C05361=1026.292,340.312,-136.892,171.555,47.662,159.342
C05362=1026.299,340.560,-136.929,171.561,47.662,159.342
C05363=1026.307,340.806,-136.966,171.568,47.662,159.343
C05364=1026.314,341.053,-137.002,171.574,47.662,159.344
C05365=1026.322,341.300,-137.038,171.581,47.662,159.345
C05366=1026.329,341.548,-137.075,171.586,47.662,159.346
C05367=1026.336,341.795,-137.111,171.593,47.661,159.347
C05368=1026.344,342.042,-137.148,171.599,47.662,159.347
C05369=1026.351,342.290,-137.185,171.606,47.661,159.348
C05370=1026.359,342.537,-137.222,171.612,47.662,159.349
C05371=1026.366,342.784,-137.259,171.618,47.661,159.350
C05372=1026.374,343.031,-137.296,171.624,47.662,159.351
C05373=1026.382,343.279,-137.332,171.631,47.662,159.352
C05374=1026.388,343.525,-137.369,171.637,47.662,159.352
C05375=1026.396,343.772,-137.405,171.644,47.662,159.353
C05376=1026.404,344.019,-137.442,171.650,47.661,159.354
C05377=1026.411,344.266,-137.480,171.657,47.662,159.355
C05378=1026.419,344.514,-137.516,171.663,47.662,159.356
C05379=1026.426,344.761,-137.554,171.669,47.661,159.357
C05380=1026.434,345.008,-137.591,171.675,47.662,159.358
C05381=1026.441,345.256,-137.627,171.682,47.662,159.359
C05382=1026.450,345.503,-137.665,171.688,47.662,159.360
C05383=1026.458,345.750,-137.702,171.695,47.662,159.360
C05384=1026.465,345.997,-137.739,171.702,47.662,159.361
C05385=1026.473,346.244,-137.776,171.708,47.662,159.362
C05386=1026.480,346.492,-137.813,171.715,47.662,159.363
C05387=1026.488,346.739,-137.850,171.721,47.663,159.364
C05388=1026.495,346.986,-137.887,171.728,47.662,159.365
C05389=1026.503,347.232,-137.924,171.735,47.662,159.366
C05390=1026.510,347.480,-137.962,171.741,47.663,159.367
C05391=1026.519,347.727,-137.999,171.748,47.663,159.368
C05392=1026.527,347.974,-138.036,171.754,47.663,159.369
C05393=1026.534,348.221,-138.074,171.761,47.663,159.370
C05394=1026.541,348.468,-138.111,171.768,47.664,159.371
C05395=1026.549,348.715,-138.148,171.774,47.664,159.371
C05396=1026.557,348.962,-138.186,171.781,47.664,159.372
C05397=1026.564,349.210,-138.223,171.787,47.664,159.373
C05398=1026.573,349.456,-138.261,171.794,47.665,159.374
C05399=1026.580,349.703,-138.299,171.801,47.665,159.375
C05400=1026.587,349.950,-138.336,171.807,47.665,159.376
C05401=1026.595,350.197,-138.373,171.814,47.666,159.377
C05402=1026.602,350.418,-138.407,171.820,47.666,159.378
C05403=1026.609,350.638,-138.441,171.826,47.666,159.379
C05404=1026.616,350.859,-138.475,171.832,47.666,159.380
C05405=1026.622,351.080,-138.508,171.838,47.667,159.381
C05406=1026.630,351.301,-138.542,171.844,47.667,159.382
C05407=1026.636,351.521,-138.576,171.850,47.667,159.383
C05408=1026.644,351.742,-138.609,171.856,47.668,159.383
C05409=1026.650,351.962,-138.643,171.863,47.668,159.384
C05410=1026.658,352.210,-138.681,171.869,47.668,159.385
C05411=1026.667,352.456,-138.719,171.876,47.668,159.386
C05412=1026.674,352.704,-138.757,171.883,47.669,159.387
C05413=1026.682,352.950,-138.795,171.889,47.669,159.388
C05414=1026.690,353.197,-138.832,171.896,47.670,159.389
C05415=1026.698,353.444,-138.870,171.903,47.670,159.390
C05416=1026.705,353.691,-138.908,171.910,47.670,159.391
C05417=1026.714,353.938,-138.946,171.916,47.671,159.392
C05418=1026.722,354.185,-138.984,171.924,47.671,159.393
C05419=1026.730,354.433,-139.022,171.931,47.672,159.394
C05420=1026.737,354.679,-139.060,171.938,47.672,159.396
C05421=1026.746,354.926,-139.098,171.944,47.673,159.396
C05422=1026.753,355.173,-139.136,171.951,47.673,159.398
C05423=1026.761,355.420,-139.175,171.959,47.674,159.399
C05424=1026.769,355.667,-139.213,171.966,47.674,159.400
C05425=1026.777,355.914,-139.251,171.972,47.675,159.401
C05426=1026.785,356.161,-139.290,171.979,47.675,159.402
C05427=1026.793,356.408,-139.328,171.986,47.676,159.403
C05428=1026.800,356.654,-139.366,171.994,47.677,159.404
C05429=1026.809,356.902,-139.405,172.001,47.677,159.405
C05430=1026.816,357.149,-139.443,172.008,47.677,159.406
C05431=1026.824,357.396,-139.481,172.014,47.678,159.407
C05432=1026.833,357.643,-139.519,172.022,47.679,159.409
C05433=1026.841,357.889,-139.558,172.029,47.680,159.410
C05434=1026.849,358.136,-139.597,172.036,47.680,159.411
C05435=1026.857,358.383,-139.635,172.043,47.680,159.412
C05436=1026.865,358.630,-139.674,172.051,47.681,159.413
C05437=1026.873,358.877,-139.712,172.057,47.682,159.414
C05438=1026.881,359.124,-139.751,172.064,47.683,159.415
C05439=1026.888,359.371,-139.789,172.072,47.684,159.416
C05440=1026.897,359.617,-139.828,172.079,47.684,159.418
C05441=1026.905,359.864,-139.867,172.086,47.685,159.419
C05442=1026.913,360.111,-139.905,172.094,47.686,159.420
C05443=1026.921,360.358,-139.944,172.101,47.686,159.421
C05444=1026.929,360.605,-139.983,172.108,47.687,159.422
C05445=1026.937,360.852,-140.022,172.116,47.688,159.423
C05446=1026.944,361.098,-140.061,172.123,47.688,159.424
C05447=1026.953,361.345,-140.100,172.129,47.689,159.426
C05448=1026.961,361.592,-140.139,172.137,47.690,159.427
C05449=1026.969,361.839,-140.178,172.144,47.691,159.428
C05450=1026.977,362.086,-140.218,172.152,47.692,159.429
C05451=1026.985,362.332,-140.257,172.159,47.693,159.430
C05452=1026.993,362.579,-140.295,172.166,47.693,159.432
C05453=1027.001,362.826,-140.335,172.174,47.695,159.433
C05454=1027.009,363.073,-140.374,172.181,47.695,159.434
C05455=1027.017,363.320,-140.413,172.189,47.696,159.435
C05456=1027.026,363.567,-140.453,172.196,47.697,159.437
C05457=1027.034,363.813,-140.492,172.203,47.698,159.438
C05458=1027.042,364.061,-140.531,172.211,47.699,159.439
C05459=1027.050,364.307,-140.570,172.218,47.700,159.440
C05460=1027.058,364.553,-140.609,172.226,47.700,159.441
C05461=1027.066,364.800,-140.649,172.233,47.702,159.443
C05462=1027.073,365.024,-140.685,172.241,47.702,159.444
C05463=1027.081,365.248,-140.720,172.247,47.703,159.445
C05464=1027.088,365.472,-140.756,172.254,47.704,159.446
C05465=1027.096,365.696,-140.792,172.261,47.705,159.447
C05466=1027.103,365.920,-140.828,172.268,47.706,159.448
C05467=1027.111,366.144,-140.863,172.274,47.707,159.449
C05468=1027.119,366.367,-140.899,172.282,47.708,159.451
C05469=1027.126,366.591,-140.935,172.288,47.709,159.452
C05470=1027.134,366.838,-140.974,172.296,47.710,159.453
C05471=1027.143,367.084,-141.014,172.303,47.711,159.454
C05472=1027.152,367.332,-141.055,172.311,47.712,159.456
C05473=1027.160,367.578,-141.094,172.319,47.712,159.457
C05474=1027.168,367.825,-141.133,172.327,47.714,159.458
C05475=1027.177,368.071,-141.173,172.335,47.715,159.460
C05476=1027.185,368.318,-141.213,172.342,47.716,159.461
C05477=1027.193,368.564,-141.253,172.350,47.717,159.462
C05478=1027.202,368.812,-141.292,172.357,47.718,159.464
C05479=1027.210,369.058,-141.332,172.366,47.719,159.465
C05480=1027.219,369.304,-141.372,172.374,47.720,159.466
C05481=1027.227,369.551,-141.412,172.381,47.722,159.468
C05482=1027.235,369.798,-141.453,172.389,47.723,159.469
C05483=1027.244,370.045,-141.493,172.397,47.724,159.470
C05484=1027.252,370.291,-141.533,172.404,47.725,159.472
C05485=1027.260,370.538,-141.573,172.413,47.726,159.473
C05486=1027.268,370.784,-141.613,172.421,47.728,159.475
C05487=1027.277,371.032,-141.653,172.428,47.729,159.476
C05488=1027.285,371.278,-141.694,172.436,47.731,159.477
C05489=1027.293,371.524,-141.734,172.444,47.732,159.479
C05490=1027.303,371.771,-141.775,172.452,47.733,159.480
C05491=1027.310,372.018,-141.814,172.460,47.734,159.482
C05492=1027.319,372.264,-141.855,172.468,47.735,159.483
C05493=1027.328,372.511,-141.896,172.476,47.737,159.484
C05494=1027.336,372.757,-141.936,172.484,47.738,159.486
C05495=1027.344,373.003,-141.975,172.492,47.739,159.487
C05496=1027.353,373.250,-142.016,172.500,47.741,159.489
C05497=1027.361,373.497,-142.057,172.509,47.742,159.490
C05498=1027.370,373.743,-142.098,172.516,47.743,159.492
C05499=1027.378,373.990,-142.138,172.524,47.745,159.493
C05500=1027.388,374.236,-142.179,172.533,47.746,159.495
C05501=1027.396,374.483,-142.219,172.541,47.747,159.496
C05502=1027.404,374.730,-142.260,172.549,47.749,159.497
C05503=1027.413,374.976,-142.300,172.557,47.750,159.499
C05504=1027.422,375.223,-142.341,172.565,47.752,159.500
C05505=1027.431,375.468,-142.381,172.573,47.753,159.502
C05506=1027.439,375.715,-142.423,172.582,47.755,159.503
C05507=1027.448,375.962,-142.464,172.590,47.757,159.505
C05508=1027.457,376.208,-142.504,172.599,47.758,159.506
C05509=1027.465,376.455,-142.545,172.607,47.759,159.508
C05510=1027.475,376.701,-142.585,172.616,47.761,159.510
C05511=1027.483,376.947,-142.627,172.623,47.762,159.511
C05512=1027.492,377.194,-142.668,172.631,47.764,159.512
C05513=1027.500,377.441,-142.709,172.640,47.766,159.514
C05514=1027.509,377.687,-142.750,172.648,47.767,159.516
C05515=1027.518,377.933,-142.792,172.657,47.769,159.517
C05516=1027.526,378.180,-142.833,172.665,47.771,159.519
C05517=1027.535,378.426,-142.874,172.674,47.772,159.520
C05518=1027.544,378.672,-142.915,172.682,47.773,159.522
C05519=1027.553,378.919,-142.956,172.691,47.775,159.523
C05520=1027.561,379.164,-142.998,172.699,47.777,159.525
C05521=1027.570,379.411,-143.039,172.708,47.778,159.527
C05522=1027.578,379.636,-143.077,172.716,47.780,159.528
C05523=1027.586,379.862,-143.115,172.724,47.782,159.530
C05524=1027.594,380.087,-143.152,172.731,47.783,159.531
C05525=1027.602,380.312,-143.191,172.739,47.785,159.533
C05526=1027.610,380.537,-143.229,172.747,47.786,159.534
C05527=1027.618,380.762,-143.266,172.755,47.788,159.535
C05528=1027.626,380.987,-143.305,172.763,47.790,159.537
C05529=1027.634,381.213,-143.343,172.771,47.791,159.538
C05530=1027.643,381.458,-143.384,172.779,47.793,159.540
C05531=1027.651,381.705,-143.426,172.788,47.795,159.542
C05532=1027.660,381.951,-143.467,172.796,47.797,159.543
C05533=1027.669,382.197,-143.509,172.805,47.799,159.545
C05534=1027.679,382.443,-143.550,172.814,47.800,159.547
C05535=1027.688,382.690,-143.592,172.822,47.802,159.548
C05536=1027.697,382.936,-143.634,172.832,47.804,159.550
C05537=1027.706,383.182,-143.676,172.841,47.806,159.552
C05538=1027.715,383.428,-143.718,172.849,47.808,159.553
C05539=1027.724,383.675,-143.760,172.858,47.810,159.555
C05540=1027.733,383.921,-143.801,172.867,47.812,159.557
C05541=1027.743,384.168,-143.844,172.876,47.813,159.559
C05542=1027.752,384.414,-143.886,172.885,47.816,159.560
C05543=1027.761,384.660,-143.928,172.894,47.817,159.562
C05544=1027.770,384.906,-143.970,172.903,47.819,159.564
C05545=1027.779,385.152,-144.012,172.912,47.821,159.566
C05546=1027.788,385.399,-144.053,172.920,47.823,159.567
C05547=1027.797,385.644,-144.096,172.930,47.825,159.569
C05548=1027.807,385.892,-144.138,172.939,47.827,159.571
C05549=1027.816,386.137,-144.180,172.948,47.829,159.573
C05550=1027.825,386.384,-144.222,172.957,47.831,159.574
C05551=1027.834,386.629,-144.264,172.967,47.833,159.576
C05552=1027.844,386.876,-144.307,172.975,47.835,159.578
C05553=1027.852,387.122,-144.350,172.984,47.837,159.580
C05554=1027.862,387.387,-144.395,172.995,47.840,159.582
C05555=1027.872,387.652,-144.442,173.004,47.842,159.583
C05556=1027.882,387.917,-144.487,173.014,47.844,159.585
C05557=1027.892,388.182,-144.533,173.025,47.847,159.588
C05558=1027.902,388.428,-144.576,173.034,47.849,159.589
C05559=1027.911,388.674,-144.618,173.043,47.851,159.591
C05560=1027.919,388.920,-144.661,173.053,47.853,159.593
C05561=1027.929,389.166,-144.704,173.061,47.855,159.595
C05562=1027.939,389.412,-144.747,173.070,47.857,159.597
C05563=1027.948,389.658,-144.789,173.080,47.860,159.599
C05564=1027.957,389.904,-144.832,173.089,47.862,159.600
C05565=1027.967,390.151,-144.875,173.099,47.864,159.602
C05566=1027.975,390.397,-144.918,173.108,47.867,159.604
C05567=1027.985,390.642,-144.961,173.118,47.869,159.606
C05568=1027.995,390.889,-145.004,173.127,47.871,159.608
C05569=1028.004,391.135,-145.048,173.137,47.873,159.610
C05570=1028.013,391.381,-145.090,173.146,47.876,159.612
C05571=1028.022,391.627,-145.134,173.156,47.878,159.614
C05572=1028.032,391.873,-145.177,173.165,47.881,159.616
C05573=1028.042,392.119,-145.220,173.176,47.882,159.618
C05574=1028.050,392.365,-145.263,173.185,47.885,159.620
C05575=1028.060,392.611,-145.307,173.195,47.888,159.622
C05576=1028.070,392.857,-145.350,173.205,47.890,159.624
C05577=1028.079,393.103,-145.393,173.214,47.892,159.626
C05578=1028.089,393.349,-145.436,173.224,47.895,159.628
C05579=1028.098,393.595,-145.480,173.233,47.897,159.630
C05580=1028.108,393.841,-145.524,173.243,47.900,159.632
C05581=1028.117,394.086,-145.567,173.254,47.902,159.634
C05582=1028.127,394.346,-145.613,173.263,47.905,159.636
C05583=1028.137,394.604,-145.659,173.274,47.907,159.638
C05584=1028.148,394.864,-145.705,173.284,47.910,159.640
C05585=1028.157,395.122,-145.751,173.295,47.913,159.642
C05586=1028.168,395.368,-145.795,173.304,47.915,159.644
C05587=1028.176,395.614,-145.839,173.314,47.918,159.646
C05588=1028.187,395.859,-145.882,173.325,47.921,159.648
C05589=1028.196,396.106,-145.926,173.335,47.923,159.650
C05590=1028.205,396.352,-145.970,173.345,47.926,159.653
C05591=1028.216,396.598,-146.014,173.355,47.928,159.655
C05592=1028.225,396.844,-146.058,173.365,47.931,159.657
C05593=1028.235,397.090,-146.102,173.375,47.934,159.659
C05594=1028.245,397.335,-146.146,173.386,47.936,159.661
C05595=1028.255,397.581,-146.190,173.395,47.939,159.663
C05596=1028.264,397.827,-146.234,173.405,47.942,159.665
C05597=1028.274,398.073,-146.278,173.416,47.944,159.667
C05598=1028.284,398.318,-146.322,173.426,47.947,159.670
C05599=1028.294,398.564,-146.366,173.437,47.950,159.672
C05600=1028.303,398.810,-146.411,173.447,47.953,159.674
C05601=1028.313,399.056,-146.455,173.456,47.955,159.676
C05602=1028.323,399.301,-146.500,173.467,47.958,159.678
C05603=1028.333,399.547,-146.544,173.477,47.961,159.680
C05604=1028.343,399.794,-146.589,173.488,47.964,159.683
C05605=1028.353,400.039,-146.633,173.498,47.967,159.685
C05606=1028.363,400.284,-146.678,173.509,47.970,159.687
C05607=1028.372,400.531,-146.722,173.519,47.973,159.689
C05608=1028.382,400.776,-146.767,173.530,47.976,159.692
C05609=1028.393,401.022,-146.812,173.540,47.979,159.694
C05610=1028.403,401.267,-146.856,173.551,47.982,159.696
C05611=1028.413,401.513,-146.901,173.561,47.985,159.698
C05612=1028.422,401.758,-146.946,173.572,47.988,159.701
C05613=1028.433,402.005,-146.991,173.583,47.990,159.703
C05614=1028.442,402.250,-147.036,173.593,47.994,159.705
C05615=1028.452,402.496,-147.081,173.604,47.996,159.707
C05616=1028.462,402.742,-147.126,173.614,47.999,159.710
C05617=1028.472,402.987,-147.171,173.625,48.002,159.712
C05618=1028.483,403.233,-147.217,173.637,48.006,159.714
C05619=1028.493,403.479,-147.262,173.647,48.009,159.717
C05620=1028.502,403.724,-147.306,173.658,48.012,159.719
C05621=1028.513,403.970,-147.352,173.669,48.015,159.721
C05622=1028.523,404.215,-147.397,173.680,48.018,159.724
C05623=1028.533,404.461,-147.442,173.691,48.021,159.726
C05624=1028.543,404.706,-147.488,173.702,48.024,159.729
C05625=1028.553,404.952,-147.533,173.713,48.028,159.731
C05626=1028.564,405.198,-147.579,173.724,48.030,159.733
C05627=1028.574,405.444,-147.624,173.734,48.034,159.736
C05628=1028.584,405.689,-147.670,173.746,48.037,159.738
C05629=1028.594,405.934,-147.715,173.757,48.040,159.741
C05630=1028.605,406.180,-147.760,173.768,48.044,159.743
C05631=1028.615,406.426,-147.806,173.780,48.047,159.746
C05632=1028.626,406.671,-147.852,173.791,48.050,159.748
C05633=1028.636,406.917,-147.897,173.802,48.053,159.750
C05634=1028.646,407.163,-147.943,173.813,48.056,159.753
C05635=1028.657,407.408,-147.989,173.825,48.060,159.755
C05636=1028.667,407.654,-148.035,173.836,48.063,159.758
C05637=1028.678,407.899,-148.081,173.848,48.066,159.760
C05638=1028.687,408.145,-148.127,173.859,48.070,159.763
C05639=1028.698,408.390,-148.173,173.870,48.073,159.765
C05640=1028.709,408.636,-148.219,173.882,48.076,159.768
C05641=1028.719,408.881,-148.265,173.893,48.080,159.770
C05642=1028.732,409.163,-148.317,173.906,48.084,159.773
C05643=1028.744,409.442,-148.370,173.919,48.088,159.776
C05644=1028.756,409.723,-148.422,173.932,48.092,159.779
C05645=1028.769,410.004,-148.475,173.946,48.095,159.782
C05646=1028.780,410.249,-148.521,173.958,48.099,159.785
C05647=1028.789,410.495,-148.568,173.969,48.103,159.787
C05648=1028.800,410.740,-148.614,173.981,48.107,159.790
C05649=1028.810,410.986,-148.661,173.992,48.110,159.793
C05650=1028.821,411.231,-148.708,174.005,48.113,159.795
C05651=1028.832,411.477,-148.754,174.017,48.117,159.798
C05652=1028.842,411.722,-148.801,174.028,48.121,159.801
C05653=1028.853,411.967,-148.847,174.040,48.124,159.803
C05654=1028.865,412.213,-148.894,174.052,48.128,159.806
C05655=1028.874,412.458,-148.941,174.064,48.132,159.809
C05656=1028.885,412.703,-148.987,174.076,48.136,159.812
C05657=1028.896,412.948,-149.034,174.088,48.140,159.814
C05658=1028.907,413.194,-149.082,174.101,48.143,159.817
C05659=1028.918,413.439,-149.128,174.112,48.147,159.820
C05660=1028.928,413.685,-149.175,174.125,48.150,159.823
C05661=1028.940,413.930,-149.222,174.137,48.154,159.825
C05662=1028.951,414.175,-149.269,174.149,48.158,159.828
C05663=1028.961,414.421,-149.317,174.161,48.162,159.831
C05664=1028.972,414.666,-149.363,174.173,48.165,159.834
C05665=1028.984,414.912,-149.410,174.186,48.169,159.836
C05666=1028.994,415.157,-149.458,174.198,48.173,159.839
C05667=1029.006,415.402,-149.505,174.211,48.177,159.842
C05668=1029.017,415.647,-149.552,174.223,48.181,159.845
C05669=1029.028,415.893,-149.600,174.235,48.185,159.848
C05670=1029.039,416.138,-149.647,174.248,48.188,159.851
C05671=1029.050,416.384,-149.694,174.260,48.193,159.854
C05672=1029.061,416.629,-149.742,174.273,48.197,159.857
C05673=1029.072,416.873,-149.790,174.285,48.200,159.859
C05674=1029.083,417.119,-149.838,174.298,48.205,159.862
C05675=1029.095,417.364,-149.885,174.311,48.209,159.865
C05676=1029.105,417.609,-149.933,174.323,48.213,159.868
C05677=1029.117,417.854,-149.981,174.337,48.217,159.871
C05678=1029.128,418.099,-150.029,174.350,48.221,159.874
C05679=1029.139,418.345,-150.077,174.362,48.224,159.877
C05680=1029.150,418.590,-150.124,174.375,48.229,159.880
C05681=1029.161,418.835,-150.172,174.388,48.233,159.883
C05682=1029.172,419.080,-150.221,174.401,48.237,159.886
C05683=1029.184,419.325,-150.268,174.414,48.241,159.889
C05684=1029.196,419.570,-150.317,174.427,48.245,159.892
C05685=1029.207,419.816,-150.366,174.440,48.249,159.895
C05686=1029.218,420.061,-150.413,174.454,48.254,159.898
C05687=1029.230,420.306,-150.462,174.467,48.258,159.901
C05688=1029.242,420.550,-150.510,174.479,48.262,159.904
C05689=1029.253,420.796,-150.558,174.493,48.267,159.908
C05690=1029.264,421.041,-150.607,174.506,48.271,159.911
C05691=1029.276,421.286,-150.655,174.520,48.275,159.914
C05692=1029.287,421.531,-150.703,174.533,48.279,159.917
C05693=1029.299,421.776,-150.752,174.547,48.284,159.920
C05694=1029.310,422.021,-150.800,174.560,48.288,159.923
C05695=1029.322,422.266,-150.850,174.574,48.293,159.927
C05696=1029.333,422.512,-150.898,174.587,48.297,159.930
C05697=1029.345,422.756,-150.947,174.600,48.301,159.933
C05698=1029.357,423.001,-150.995,174.614,48.306,159.936
C05699=1029.369,423.246,-151.045,174.628,48.310,159.939
C05700=1029.380,423.491,-151.094,174.642,48.314,159.943
C05701=1029.392,423.736,-151.143,174.655,48.319,159.946
C05702=1029.406,424.027,-151.201,174.672,48.325,159.950
C05703=1029.420,424.318,-151.260,174.688,48.330,159.954
C05704=1029.434,424.609,-151.318,174.704,48.335,159.957
C05705=1029.448,424.900,-151.376,174.721,48.341,159.961
C05706=1029.460,425.145,-151.425,174.736,48.345,159.965
C05707=1029.472,425.390,-151.475,174.749,48.350,159.968
C05708=1029.483,425.634,-151.525,174.764,48.355,159.972
C05709=1029.495,425.880,-151.574,174.777,48.359,159.975
C05710=1029.508,426.123,-151.623,174.792,48.364,159.978
C05711=1029.520,426.369,-151.672,174.806,48.369,159.982
C05712=1029.532,426.614,-151.722,174.821,48.373,159.985
C05713=1029.543,426.858,-151.772,174.834,48.378,159.989
C05714=1029.556,427.103,-151.822,174.849,48.383,159.992
C05715=1029.567,427.348,-151.872,174.863,48.388,159.995
C05716=1029.579,427.592,-151.922,174.878,48.392,159.999
C05717=1029.591,427.838,-151.971,174.893,48.397,160.002
C05718=1029.603,428.083,-152.022,174.907,48.402,160.006
C05719=1029.616,428.328,-152.072,174.921,48.407,160.009
C05720=1029.627,428.572,-152.121,174.937,48.412,160.013
C05721=1029.640,428.816,-152.171,174.952,48.416,160.017
C05722=1029.652,429.061,-152.222,174.965,48.421,160.020
C05723=1029.665,429.306,-152.272,174.981,48.427,160.024
C05724=1029.676,429.551,-152.323,174.995,48.431,160.027
C05725=1029.688,429.795,-152.373,175.011,48.436,160.031
C05726=1029.701,430.040,-152.424,175.025,48.441,160.035
C05727=1029.713,430.284,-152.474,175.041,48.446,160.038
C05728=1029.726,430.529,-152.525,175.056,48.451,160.042
C05729=1029.738,430.774,-152.575,175.071,48.456,160.046
C05730=1029.751,431.018,-152.626,175.086,48.461,160.049
C05731=1029.763,431.263,-152.676,175.101,48.466,160.053
C05732=1029.776,431.507,-152.727,175.116,48.471,160.057
C05733=1029.789,431.751,-152.777,175.132,48.477,160.060
C05734=1029.801,431.996,-152.828,175.147,48.482,160.064
C05735=1029.813,432.241,-152.879,175.162,48.487,160.068
C05736=1029.826,432.485,-152.930,175.178,48.492,160.072
C05737=1029.839,432.729,-152.981,175.193,48.497,160.075
C05738=1029.852,432.974,-153.032,175.209,48.502,160.079
C05739=1029.864,433.218,-153.083,175.225,48.507,160.083
C05740=1029.878,433.463,-153.134,175.240,48.512,160.087
C05741=1029.890,433.708,-153.185,175.256,48.518,160.091
C05742=1029.902,433.952,-153.236,175.272,48.523,160.095
C05743=1029.915,434.197,-153.287,175.288,48.528,160.099
C05744=1029.928,434.441,-153.339,175.304,48.534,160.103
C05745=1029.941,434.686,-153.391,175.320,48.539,160.106
C05746=1029.954,434.929,-153.442,175.335,48.544,160.110
C05747=1029.967,435.174,-153.493,175.352,48.550,160.114
C05748=1029.980,435.418,-153.545,175.367,48.555,160.118
C05749=1029.993,435.662,-153.598,175.384,48.561,160.122
C05750=1030.006,435.907,-153.649,175.401,48.566,160.126
C05751=1030.019,436.151,-153.700,175.416,48.571,160.130
C05752=1030.032,436.396,-153.753,175.433,48.577,160.134
C05753=1030.045,436.640,-153.805,175.450,48.582,160.138
C05754=1030.057,436.884,-153.857,175.465,48.588,160.142
C05755=1030.071,437.128,-153.909,175.482,48.594,160.147
C05756=1030.084,437.372,-153.961,175.499,48.599,160.151
C05757=1030.097,437.617,-154.013,175.516,48.605,160.155
C05758=1030.111,437.861,-154.065,175.533,48.611,160.159
C05759=1030.123,438.104,-154.118,175.550,48.616,160.163
C05760=1030.137,438.349,-154.170,175.566,48.622,160.167
C05761=1030.150,438.593,-154.222,175.582,48.628,160.172
C05762=1030.165,438.860,-154.279,175.602,48.633,160.176
C05763=1030.179,439.127,-154.337,175.620,48.640,160.181
C05764=1030.195,439.394,-154.395,175.639,48.646,160.186
C05765=1030.208,439.660,-154.452,175.657,48.652,160.190
C05766=1030.223,439.905,-154.505,175.675,48.658,160.195
C05767=1030.236,440.149,-154.557,175.692,48.664,160.199
C05768=1030.249,440.393,-154.610,175.709,48.670,160.203
C05769=1030.263,440.637,-154.663,175.727,48.676,160.208
C05770=1030.276,440.880,-154.716,175.744,48.681,160.212
C05771=1030.290,441.125,-154.769,175.761,48.688,160.216
C05772=1030.304,441.369,-154.822,175.780,48.694,160.221
C05773=1030.317,441.613,-154.875,175.797,48.699,160.225
C05774=1030.332,441.857,-154.929,175.815,48.705,160.229
C05775=1030.345,442.100,-154.982,175.832,48.711,160.234
C05776=1030.359,442.344,-155.035,175.851,48.717,160.238
C05777=1030.373,442.588,-155.089,175.868,48.723,160.243
C05778=1030.387,442.832,-155.142,175.886,48.729,160.247
C05779=1030.401,443.075,-155.195,175.904,48.735,160.252
C05780=1030.415,443.318,-155.248,175.922,48.741,160.256
C05781=1030.429,443.562,-155.301,175.941,48.747,160.261
C05782=1030.444,443.804,-155.354,175.959,48.753,160.266
C05783=1030.459,444.048,-155.405,175.977,48.758,160.270
C05784=1030.476,444.291,-155.456,175.996,48.764,160.275
C05785=1030.492,444.535,-155.508,176.014,48.770,160.279
C05786=1030.509,444.778,-155.559,176.032,48.776,160.284
C05787=1030.527,445.023,-155.609,176.052,48.781,160.288
C05788=1030.544,445.266,-155.659,176.070,48.787,160.293
C05789=1030.564,445.511,-155.708,176.089,48.792,160.297
C05790=1030.582,445.754,-155.758,176.107,48.797,160.302
C05791=1030.602,445.999,-155.807,176.126,48.802,160.306
C05792=1030.622,446.243,-155.854,176.146,48.807,160.310
C05793=1030.642,446.488,-155.902,176.164,48.812,160.315
C05794=1030.663,446.732,-155.950,176.184,48.817,160.319
C05795=1030.685,446.976,-155.997,176.204,48.822,160.324
C05796=1030.706,447.220,-156.044,176.223,48.827,160.328
C05797=1030.729,447.466,-156.090,176.242,48.832,160.333
C05798=1030.751,447.710,-156.136,176.262,48.836,160.337
C05799=1030.775,447.954,-156.181,176.282,48.841,160.341
C05800=1030.799,448.199,-156.226,176.301,48.845,160.346
C05801=1030.823,448.444,-156.271,176.321,48.850,160.350
C05802=1030.848,448.689,-156.315,176.341,48.855,160.355
C05803=1030.873,448.934,-156.358,176.361,48.859,160.359
C05804=1030.899,449.179,-156.402,176.382,48.863,160.363
C05805=1030.926,449.424,-156.445,176.402,48.867,160.368
C05806=1030.953,449.669,-156.488,176.421,48.871,160.372
C05807=1030.979,449.914,-156.530,176.442,48.875,160.377
C05808=1031.008,450.159,-156.571,176.463,48.879,160.381
C05809=1031.036,450.404,-156.612,176.483,48.883,160.385
C05810=1031.064,450.650,-156.653,176.504,48.887,160.390
C05811=1031.094,450.896,-156.694,176.524,48.891,160.394
C05812=1031.124,451.141,-156.734,176.545,48.895,160.398
C05813=1031.154,451.386,-156.774,176.566,48.898,160.403
C05814=1031.185,451.632,-156.813,176.588,48.902,160.407
C05815=1031.215,451.878,-156.852,176.608,48.905,160.411
C05816=1031.247,452.124,-156.890,176.629,48.909,160.416
C05817=1031.279,452.369,-156.928,176.651,48.912,160.420
C05818=1031.312,452.615,-156.966,176.672,48.915,160.424
C05819=1031.345,452.860,-157.003,176.693,48.919,160.429
C05820=1031.379,453.106,-157.039,176.714,48.922,160.433
C05821=1031.414,453.351,-157.076,176.736,48.925,160.437
C05822=1031.446,453.582,-157.110,176.756,48.928,160.441
C05823=1031.165,453.651,-157.442,176.760,48.992,160.462
C05824=1031.139,453.464,-157.415,176.743,48.990,160.459
C05825=1031.104,453.218,-157.379,176.721,48.986,160.454
C05826=1031.070,452.973,-157.342,176.700,48.984,160.450
C05827=1031.037,452.727,-157.306,176.678,48.981,160.446
C05828=1031.004,452.481,-157.267,176.658,48.977,160.441
C05829=1030.972,452.236,-157.230,176.636,48.974,160.437
C05830=1030.939,451.991,-157.192,176.614,48.971,160.433
C05831=1030.908,451.745,-157.153,176.593,48.967,160.428
C05832=1030.877,451.498,-157.114,176.572,48.964,160.424
C05833=1030.847,451.254,-157.075,176.551,48.960,160.420
C05834=1030.817,451.008,-157.036,176.531,48.957,160.415
C05835=1030.787,450.762,-156.995,176.510,48.953,160.411
C05836=1030.758,450.517,-156.954,176.489,48.949,160.407
C05837=1030.730,450.272,-156.914,176.468,48.946,160.402
C05838=1030.702,450.027,-156.872,176.447,48.942,160.398
C05839=1030.674,449.781,-156.830,176.427,48.937,160.394
C05840=1030.647,449.536,-156.787,176.407,48.933,160.389
C05841=1030.620,449.291,-156.745,176.387,48.929,160.385
C05842=1030.594,449.046,-156.702,176.366,48.926,160.381
C05843=1030.569,448.801,-156.659,176.346,48.921,160.376
C05844=1030.544,448.556,-156.614,176.326,48.917,160.372
C05845=1030.519,448.311,-156.570,176.306,48.913,160.367
C05846=1030.495,448.066,-156.526,176.286,48.909,160.363
C05847=1030.471,447.821,-156.480,176.266,48.904,160.359
C05848=1030.448,447.577,-156.434,176.247,48.899,160.354
C05849=1030.426,447.332,-156.389,176.227,48.895,160.350
C05850=1030.404,447.087,-156.342,176.208,48.890,160.345
C05851=1030.382,446.843,-156.295,176.188,48.885,160.341
C05852=1030.360,446.599,-156.248,176.169,48.880,160.336
C05853=1030.339,446.354,-156.201,176.150,48.875,160.332
C05854=1030.319,446.111,-156.152,176.131,48.871,160.328
C05855=1030.299,445.866,-156.104,176.112,48.865,160.323
C05856=1030.280,445.622,-156.055,176.093,48.860,160.319
C05857=1030.262,445.378,-156.005,176.073,48.855,160.314
C05858=1030.243,445.134,-155.956,176.055,48.850,160.310
C05859=1030.225,444.890,-155.906,176.036,48.845,160.305
C05860=1030.208,444.647,-155.856,176.018,48.839,160.301
C05861=1030.191,444.402,-155.805,175.999,48.834,160.296
C05862=1030.175,444.159,-155.753,175.980,48.828,160.292
C05863=1030.159,443.915,-155.702,175.962,48.823,160.287
C05864=1030.144,443.672,-155.649,175.943,48.817,160.283
C05865=1030.128,443.428,-155.597,175.925,48.811,160.278
C05866=1030.114,443.185,-155.544,175.907,48.805,160.274
C05867=1030.100,442.942,-155.490,175.889,48.799,160.269
C05868=1030.086,442.699,-155.438,175.871,48.793,160.265
C05869=1030.072,442.456,-155.384,175.853,48.787,160.260
C05870=1030.059,442.212,-155.331,175.835,48.781,160.256
C05871=1030.044,441.968,-155.277,175.817,48.776,160.251
C05872=1030.031,441.724,-155.224,175.800,48.770,160.247
C05873=1030.017,441.480,-155.171,175.781,48.764,160.242
C05874=1030.004,441.236,-155.118,175.764,48.758,160.238
C05875=1029.990,440.992,-155.065,175.746,48.753,160.233
C05876=1029.976,440.748,-155.013,175.729,48.747,160.229
C05877=1029.962,440.504,-154.959,175.712,48.741,160.225
C05878=1029.949,440.260,-154.907,175.694,48.735,160.220
C05879=1029.935,440.016,-154.853,175.677,48.730,160.216
C05880=1029.922,439.772,-154.801,175.660,48.724,160.212
C05881=1029.907,439.504,-154.743,175.641,48.717,160.207
C05882=1029.893,439.236,-154.685,175.621,48.711,160.202
C05883=1029.878,438.968,-154.627,175.603,48.705,160.198
C05884=1029.864,438.701,-154.570,175.584,48.699,160.193
C05885=1029.850,438.457,-154.518,175.567,48.693,160.189
C05886=1029.836,438.213,-154.465,175.551,48.688,160.185
C05887=1029.824,437.969,-154.413,175.534,48.682,160.180
C05888=1029.810,437.724,-154.361,175.517,48.677,160.176
C05889=1029.797,437.480,-154.309,175.500,48.671,160.172
C05890=1029.784,437.235,-154.256,175.483,48.666,160.168
C05891=1029.771,436.992,-154.205,175.466,48.660,160.164
C05892=1029.758,436.747,-154.152,175.451,48.655,160.160
C05893=1029.744,436.503,-154.100,175.434,48.650,160.156
C05894=1029.731,436.259,-154.049,175.417,48.644,160.152
C05895=1029.719,436.015,-153.996,175.400,48.639,160.148
C05896=1029.705,435.771,-153.945,175.385,48.633,160.144
C05897=1029.692,435.526,-153.893,175.368,48.628,160.140
C05898=1029.680,435.282,-153.841,175.352,48.623,160.136
C05899=1029.666,435.037,-153.789,175.336,48.617,160.132
C05900=1029.654,434.793,-153.739,175.320,48.612,160.128
C05901=1029.640,434.549,-153.687,175.304,48.606,160.124
C05902=1029.628,434.304,-153.635,175.288,48.602,160.120
C05903=1029.615,434.060,-153.583,175.272,48.596,160.116
C05904=1029.602,433.816,-153.533,175.256,48.591,160.112
C05905=1029.590,433.571,-153.481,175.240,48.586,160.108
C05906=1029.577,433.327,-153.430,175.225,48.581,160.105
C05907=1029.564,433.082,-153.379,175.209,48.576,160.101
C05908=1029.551,432.837,-153.328,175.193,48.570,160.097
C05909=1029.539,432.593,-153.277,175.178,48.565,160.093
C05910=1029.526,432.349,-153.226,175.162,48.560,160.089
C05911=1029.513,432.104,-153.175,175.147,48.555,160.086
C05912=1029.500,431.860,-153.124,175.131,48.550,160.082
C05913=1029.488,431.615,-153.074,175.116,48.545,160.078
C05914=1029.475,431.371,-153.023,175.100,48.540,160.074
C05915=1029.463,431.127,-152.973,175.085,48.536,160.071
C05916=1029.450,430.881,-152.922,175.070,48.530,160.067
C05917=1029.438,430.637,-152.871,175.054,48.525,160.063
C05918=1029.425,430.392,-152.821,175.040,48.521,160.060
C05919=1029.413,430.148,-152.770,175.024,48.516,160.056
C05920=1029.401,429.903,-152.720,175.009,48.511,160.052
C05921=1029.388,429.658,-152.670,174.994,48.506,160.049
C05922=1029.376,429.415,-152.619,174.979,48.501,160.045
C05923=1029.364,429.170,-152.569,174.964,48.496,160.041
C05924=1029.352,428.925,-152.519,174.950,48.491,160.038
C05925=1029.339,428.680,-152.469,174.935,48.486,160.034
C05926=1029.327,428.435,-152.419,174.921,48.482,160.031
C05927=1029.315,428.190,-152.368,174.906,48.477,160.027
C05928=1029.304,427.946,-152.318,174.891,48.472,160.024
C05929=1029.291,427.701,-152.268,174.877,48.467,160.020
C05930=1029.279,427.456,-152.218,174.862,48.463,160.017
C05931=1029.267,427.212,-152.168,174.847,48.458,160.013
C05932=1029.255,426.967,-152.118,174.833,48.453,160.010
C05933=1029.243,426.722,-152.069,174.818,48.448,160.006
C05934=1029.231,426.478,-152.019,174.804,48.444,160.003
C05935=1029.219,426.232,-151.970,174.790,48.439,160.000
C05936=1029.207,425.988,-151.920,174.775,48.435,159.996
C05937=1029.196,425.743,-151.871,174.762,48.430,159.993
C05938=1029.183,425.498,-151.821,174.747,48.426,159.989
C05939=1029.171,425.254,-151.772,174.733,48.421,159.986
C05940=1029.159,425.008,-151.723,174.719,48.417,159.983
C05941=1029.145,424.715,-151.663,174.702,48.411,159.979
C05942=1029.131,424.421,-151.605,174.686,48.406,159.975
C05943=1029.116,424.128,-151.545,174.668,48.401,159.971
C05944=1029.103,423.835,-151.487,174.652,48.396,159.967
C05945=1029.091,423.590,-151.438,174.639,48.391,159.964
C05946=1029.079,423.345,-151.389,174.625,48.387,159.961
C05947=1029.068,423.100,-151.340,174.611,48.382,159.957
C05948=1029.057,422.856,-151.291,174.597,48.378,159.954
C05949=1029.044,422.610,-151.243,174.584,48.373,159.951
C05950=1029.033,422.365,-151.194,174.570,48.369,159.948
C05951=1029.021,422.120,-151.145,174.556,48.365,159.945
C05952=1029.010,421.875,-151.096,174.542,48.361,159.941
C05953=1028.998,421.630,-151.048,174.529,48.356,159.938
C05954=1028.986,421.384,-150.999,174.516,48.352,159.935
C05955=1028.974,421.140,-150.951,174.502,48.348,159.932
C05956=1028.963,420.895,-150.903,174.489,48.344,159.929
C05957=1028.952,420.650,-150.854,174.476,48.340,159.926
C05958=1028.940,420.405,-150.806,174.463,48.335,159.923
C05959=1028.929,420.159,-150.758,174.449,48.331,159.920
C05960=1028.918,419.914,-150.709,174.436,48.327,159.916
C05961=1028.906,419.670,-150.661,174.423,48.323,159.913
C05962=1028.894,419.424,-150.612,174.410,48.319,159.910
C05963=1028.883,419.179,-150.565,174.397,48.315,159.907
C05964=1028.872,418.934,-150.516,174.383,48.311,159.904
C05965=1028.861,418.689,-150.469,174.370,48.307,159.901
C05966=1028.849,418.444,-150.421,174.357,48.303,159.898
C05967=1028.838,418.199,-150.373,174.345,48.298,159.895
C05968=1028.827,417.953,-150.324,174.332,48.295,159.892
C05969=1028.815,417.708,-150.277,174.319,48.291,159.889
C05970=1028.805,417.463,-150.229,174.306,48.287,159.886
C05971=1028.793,417.218,-150.182,174.293,48.283,159.883
C05972=1028.782,416.973,-150.133,174.281,48.279,159.881
C05973=1028.772,416.727,-150.086,174.268,48.275,159.878
C05974=1028.760,416.482,-150.038,174.255,48.272,159.875
C05975=1028.750,416.238,-149.990,174.243,48.267,159.872
C05976=1028.738,415.992,-149.944,174.230,48.264,159.869
C05977=1028.727,415.746,-149.896,174.217,48.260,159.866
C05978=1028.716,415.502,-149.849,174.206,48.256,159.863
C05979=1028.704,415.256,-149.802,174.193,48.252,159.861
C05980=1028.694,415.011,-149.754,174.181,48.248,159.858
C05981=1028.683,414.765,-149.707,174.168,48.244,159.855
C05982=1028.671,414.521,-149.660,174.156,48.241,159.852
C05983=1028.661,414.275,-149.612,174.143,48.237,159.849
C05984=1028.650,414.030,-149.566,174.132,48.233,159.846
C05985=1028.638,413.784,-149.519,174.119,48.230,159.844
C05986=1028.628,413.539,-149.472,174.107,48.226,159.841
C05987=1028.617,413.294,-149.425,174.094,48.222,159.838
C05988=1028.606,413.048,-149.377,174.083,48.219,159.835
C05989=1028.595,412.803,-149.331,174.070,48.215,159.833
C05990=1028.585,412.557,-149.285,174.058,48.211,159.830
C05991=1028.575,412.312,-149.238,174.047,48.208,159.827
C05992=1028.563,412.066,-149.191,174.034,48.204,159.825
C05993=1028.552,411.821,-149.144,174.022,48.201,159.822
C05994=1028.542,411.575,-149.098,174.011,48.197,159.819
C05995=1028.531,411.330,-149.051,173.998,48.194,159.817
C05996=1028.520,411.085,-149.004,173.986,48.190,159.814
C05997=1028.510,410.840,-148.958,173.975,48.187,159.811
C05998=1028.500,410.595,-148.911,173.963,48.183,159.809
C05999=1028.489,410.349,-148.865,173.952,48.179,159.806
C06000=1028.478,410.103,-148.818,173.939,48.176,159.803
C06001=1028.466,409.820,-148.765,173.926,48.172,159.800
C06002=1028.453,409.537,-148.712,173.913,48.168,159.797
C06003=1028.441,409.254,-148.659,173.899,48.164,159.794
C06004=1028.429,408.971,-148.605,173.886,48.161,159.792
C06005=1028.419,408.726,-148.560,173.875,48.157,159.789
C06006=1028.408,408.481,-148.514,173.863,48.154,159.787
C06007=1028.397,408.235,-148.468,173.851,48.151,159.784
C06008=1028.387,407.990,-148.422,173.840,48.148,159.781
C06009=1028.376,407.744,-148.376,173.828,48.145,159.779
C06010=1028.365,407.498,-148.330,173.817,48.141,159.776
C06011=1028.355,407.253,-148.284,173.805,48.138,159.774
C06012=1028.345,407.007,-148.239,173.794,48.135,159.771
C06013=1028.335,406.762,-148.194,173.783,48.131,159.769
C06014=1028.324,406.516,-148.148,173.772,48.128,159.767
C06015=1028.313,406.271,-148.102,173.760,48.125,159.764
C06016=1028.304,406.025,-148.057,173.750,48.121,159.762
C06017=1028.293,405.779,-148.011,173.739,48.119,159.759
C06018=1028.282,405.534,-147.965,173.727,48.115,159.757
C06019=1028.273,405.288,-147.920,173.716,48.113,159.754
C06020=1028.262,405.043,-147.875,173.705,48.109,159.752
C06021=1028.252,404.797,-147.829,173.694,48.106,159.750
C06022=1028.242,404.552,-147.784,173.682,48.103,159.747
C06023=1028.231,404.305,-147.739,173.672,48.100,159.745
C06024=1028.221,404.061,-147.693,173.661,48.097,159.743
C06025=1028.211,403.814,-147.648,173.650,48.094,159.740
C06026=1028.201,403.569,-147.603,173.639,48.091,159.738
C06027=1028.191,403.324,-147.558,173.629,48.088,159.735
C06028=1028.181,403.078,-147.512,173.618,48.085,159.733
C06029=1028.171,402.832,-147.468,173.606,48.082,159.731
C06030=1028.161,402.586,-147.422,173.595,48.079,159.728
C06031=1028.151,402.341,-147.378,173.585,48.076,159.726
C06032=1028.141,402.095,-147.333,173.574,48.073,159.724
C06033=1028.131,401.849,-147.287,173.563,48.070,159.721
C06034=1028.121,401.603,-147.243,173.553,48.067,159.719
C06035=1028.112,401.358,-147.198,173.542,48.064,159.717
C06036=1028.101,401.112,-147.153,173.532,48.061,159.715
C06037=1028.092,400.866,-147.108,173.521,48.059,159.713
C06038=1028.081,400.621,-147.064,173.510,48.056,159.710
C06039=1028.071,400.375,-147.019,173.500,48.053,159.708
C06040=1028.062,400.130,-146.974,173.489,48.050,159.706
C06041=1028.052,399.883,-146.929,173.480,48.048,159.704
C06042=1028.042,399.637,-146.885,173.469,48.045,159.701
C06043=1028.032,399.392,-146.840,173.458,48.042,159.699
C06044=1028.022,399.146,-146.796,173.448,48.039,159.697
C06045=1028.012,398.901,-146.751,173.438,48.036,159.695
C06046=1028.003,398.654,-146.707,173.427,48.034,159.693
C06047=1027.993,398.409,-146.663,173.417,48.031,159.690
C06048=1027.983,398.163,-146.619,173.406,48.029,159.688
C06049=1027.973,397.917,-146.576,173.396,48.025,159.686
C06050=1027.963,397.672,-146.531,173.386,48.023,159.684
C06051=1027.954,397.426,-146.487,173.376,48.021,159.682
C06052=1027.944,397.180,-146.443,173.366,48.018,159.680
C06053=1027.934,396.934,-146.399,173.355,48.015,159.678
C06054=1027.924,396.688,-146.355,173.345,48.013,159.676
C06055=1027.915,396.442,-146.311,173.335,48.010,159.673
C06056=1027.904,396.197,-146.267,173.325,48.008,159.671
C06057=1027.895,395.950,-146.223,173.315,48.005,159.669
C06058=1027.886,395.704,-146.179,173.305,48.003,159.667
C06059=1027.875,395.458,-146.135,173.295,48.000,159.665
C06060=1027.867,395.213,-146.092,173.285,47.998,159.663
C06061=1027.856,394.951,-146.046,173.274,47.995,159.661
C06062=1027.846,394.690,-145.998,173.264,47.993,159.659
C06063=1027.836,394.429,-145.953,173.254,47.989,159.657
C06064=1027.826,394.169,-145.906,173.243,47.987,159.655
C06065=1027.816,393.922,-145.862,173.233,47.985,159.652
C06066=1027.806,393.676,-145.819,173.223,47.982,159.650
C06067=1027.797,393.430,-145.775,173.213,47.980,159.649
C06068=1027.787,393.185,-145.732,173.203,47.978,159.647
C06069=1027.778,392.938,-145.689,173.194,47.975,159.644
C06070=1027.768,392.692,-145.645,173.184,47.973,159.643
C06071=1027.759,392.446,-145.602,173.175,47.970,159.641
C06072=1027.750,392.200,-145.558,173.165,47.968,159.639
C06073=1027.740,391.954,-145.516,173.155,47.966,159.637
C06074=1027.730,391.709,-145.472,173.145,47.963,159.635
C06075=1027.721,391.462,-145.429,173.136,47.961,159.633
C06076=1027.712,391.216,-145.387,173.126,47.959,159.631
C06077=1027.702,390.970,-145.343,173.117,47.957,159.629
C06078=1027.693,390.724,-145.300,173.107,47.955,159.627
C06079=1027.683,390.478,-145.257,173.098,47.952,159.625
C06080=1027.675,390.232,-145.214,173.088,47.950,159.623
C06081=1027.665,389.986,-145.171,173.079,47.948,159.621
C06082=1027.655,389.740,-145.128,173.069,47.946,159.620
C06083=1027.647,389.494,-145.085,173.060,47.943,159.618
C06084=1027.637,389.248,-145.042,173.050,47.941,159.616
C06085=1027.628,389.002,-145.000,173.041,47.939,159.614
C06086=1027.618,388.756,-144.957,173.032,47.937,159.612
C06087=1027.610,388.509,-144.914,173.022,47.935,159.610
C06088=1027.600,388.264,-144.872,173.013,47.933,159.608
C06089=1027.590,388.017,-144.829,173.004,47.931,159.607
C06090=1027.581,387.772,-144.787,172.994,47.929,159.605
C06091=1027.573,387.525,-144.744,172.985,47.927,159.603
C06092=1027.563,387.278,-144.701,172.976,47.925,159.601
C06093=1027.554,387.033,-144.659,172.966,47.923,159.599
C06094=1027.545,386.787,-144.617,172.957,47.921,159.597
C06095=1027.536,386.541,-144.575,172.949,47.919,159.596
C06096=1027.527,386.294,-144.531,172.940,47.917,159.594
C06097=1027.518,386.047,-144.490,172.930,47.915,159.592
C06098=1027.509,385.802,-144.447,172.921,47.913,159.590
C06099=1027.499,385.556,-144.406,172.912,47.911,159.589
C06100=1027.489,385.309,-144.363,172.903,47.909,159.587
C06101=1027.480,385.063,-144.322,172.893,47.907,159.585
C06102=1027.471,384.817,-144.279,172.885,47.906,159.584
C06103=1027.462,384.571,-144.238,172.876,47.903,159.582
C06104=1027.453,384.324,-144.196,172.867,47.902,159.580
C06105=1027.444,384.079,-144.153,172.858,47.900,159.578
C06106=1027.435,383.832,-144.112,172.849,47.898,159.577
C06107=1027.425,383.585,-144.070,172.840,47.896,159.575
C06108=1027.416,383.339,-144.028,172.831,47.895,159.573
C06109=1027.407,383.092,-143.986,172.822,47.893,159.571
C06110=1027.398,382.847,-143.944,172.813,47.891,159.570
C06111=1027.389,382.600,-143.902,172.805,47.889,159.568
C06112=1027.380,382.354,-143.860,172.796,47.888,159.567
C06113=1027.371,382.108,-143.819,172.787,47.886,159.565
C06114=1027.362,381.861,-143.777,172.779,47.884,159.563
C06115=1027.354,381.616,-143.736,172.770,47.882,159.562
C06116=1027.345,381.369,-143.694,172.761,47.881,159.560
C06117=1027.337,381.133,-143.654,172.752,47.879,159.558
C06118=1027.328,380.898,-143.615,172.744,47.877,159.557
C06119=1027.320,380.662,-143.575,172.735,47.876,159.555
C06120=1027.311,380.427,-143.534,172.727,47.874,159.554
C06121=1027.303,380.191,-143.495,172.719,47.872,159.552
C06122=1027.294,379.956,-143.456,172.711,47.871,159.551
C06123=1027.286,379.720,-143.416,172.703,47.870,159.549
C06124=1027.277,379.484,-143.376,172.695,47.868,159.548
C06125=1027.269,379.238,-143.335,172.686,47.866,159.546
C06126=1027.260,378.992,-143.293,172.678,47.864,159.544
C06127=1027.251,378.745,-143.252,172.669,47.863,159.543
C06128=1027.242,378.499,-143.210,172.661,47.861,159.541
C06129=1027.234,378.252,-143.170,172.652,47.860,159.540
C06130=1027.225,378.006,-143.128,172.644,47.858,159.538
C06131=1027.217,377.760,-143.086,172.635,47.857,159.537
C06132=1027.208,377.514,-143.046,172.627,47.855,159.535
C06133=1027.199,377.267,-143.005,172.618,47.854,159.533
C06134=1027.190,377.020,-142.964,172.610,47.852,159.532
C06135=1027.182,376.774,-142.923,172.601,47.851,159.530
C06136=1027.173,376.527,-142.883,172.593,47.849,159.529
C06137=1027.164,376.281,-142.841,172.585,47.848,159.527
C06138=1027.156,376.035,-142.800,172.577,47.846,159.526
C06139=1027.147,375.788,-142.760,172.568,47.845,159.524
C06140=1027.138,375.542,-142.719,172.560,47.843,159.523
C06141=1027.130,375.295,-142.678,172.551,47.843,159.521
C06142=1027.120,375.048,-142.638,172.543,47.841,159.520
C06143=1027.112,374.802,-142.597,172.535,47.840,159.518
C06144=1027.103,374.555,-142.557,172.527,47.839,159.517
C06145=1027.095,374.309,-142.516,172.519,47.837,159.516
C06146=1027.086,374.062,-142.475,172.510,47.836,159.514
C06147=1027.078,373.816,-142.435,172.503,47.835,159.513
C06148=1027.069,373.569,-142.394,172.494,47.833,159.511
C06149=1027.062,373.357,-142.360,172.487,47.832,159.510
C06150=1027.054,373.145,-142.325,172.480,47.831,159.509
C06151=1027.047,372.933,-142.289,172.473,47.830,159.508
C06152=1027.040,372.721,-142.255,172.467,47.828,159.506
C06153=1027.032,372.509,-142.220,172.459,47.828,159.505
C06154=1027.025,372.296,-142.186,172.453,47.826,159.504
C06155=1027.018,372.084,-142.151,172.445,47.826,159.503
C06156=1027.011,371.872,-142.116,172.439,47.825,159.502
C06157=1027.002,371.626,-142.076,172.431,47.823,159.500
C06158=1026.994,371.379,-142.035,172.422,47.822,159.499
C06159=1026.985,371.132,-141.995,172.415,47.821,159.497
C06160=1026.977,370.886,-141.955,172.407,47.819,159.496
C06161=1026.969,370.639,-141.914,172.398,47.819,159.494
C06162=1026.960,370.392,-141.875,172.391,47.817,159.493
C06163=1026.952,370.146,-141.834,172.383,47.816,159.492
C06164=1026.944,369.899,-141.794,172.375,47.815,159.490
C06165=1026.935,369.653,-141.754,172.368,47.814,159.489
C06166=1026.927,369.406,-141.714,172.359,47.813,159.488
C06167=1026.918,369.159,-141.674,172.352,47.812,159.486
C06168=1026.910,368.913,-141.634,172.344,47.811,159.485
C06169=1026.901,368.667,-141.594,172.336,47.809,159.484
C06170=1026.894,368.420,-141.554,172.328,47.808,159.482
C06171=1026.885,368.173,-141.515,172.320,47.808,159.481
C06172=1026.876,367.926,-141.475,172.313,47.807,159.480
C06173=1026.868,367.679,-141.436,172.305,47.805,159.478
C06174=1026.860,367.432,-141.396,172.298,47.805,159.477
C06175=1026.851,367.186,-141.356,172.290,47.803,159.476
C06176=1026.843,366.940,-141.316,172.281,47.802,159.474
C06177=1026.834,366.693,-141.277,172.274,47.802,159.473
C06178=1026.827,366.446,-141.237,172.266,47.801,159.472
C06179=1026.818,366.200,-141.198,172.259,47.800,159.471
C06180=1026.810,365.953,-141.158,172.251,47.799,159.469
C06181=1026.800,365.680,-141.115,172.243,47.798,159.468
C06182=1026.791,365.408,-141.071,172.234,47.797,159.467
C06183=1026.782,365.136,-141.028,172.227,47.796,159.465
C06184=1026.774,364.864,-140.985,172.218,47.795,159.464
C06185=1026.765,364.618,-140.946,172.210,47.794,159.463
C06186=1026.757,364.371,-140.906,172.203,47.793,159.461
C06187=1026.749,364.124,-140.867,172.196,47.792,159.460
C06188=1026.740,363.878,-140.827,172.188,47.791,159.459
C06189=1026.732,363.631,-140.789,172.181,47.791,159.458
C06190=1026.725,363.384,-140.749,172.172,47.790,159.456
C06191=1026.716,363.137,-140.709,172.165,47.790,159.455
C06192=1026.708,362.890,-140.670,172.157,47.788,159.454
C06193=1026.700,362.643,-140.631,172.150,47.788,159.453
C06194=1026.692,362.396,-140.592,172.143,47.787,159.452
C06195=1026.684,362.150,-140.553,172.135,47.786,159.450
C06196=1026.676,361.903,-140.514,172.128,47.786,159.449
C06197=1026.667,361.657,-140.475,172.121,47.785,159.448
C06198=1026.660,361.409,-140.435,172.113,47.784,159.447
C06199=1026.652,361.163,-140.397,172.107,47.783,159.446
C06200=1026.644,360.916,-140.358,172.099,47.782,159.444
C06201=1026.635,360.669,-140.319,172.092,47.781,159.443
C06202=1026.627,360.422,-140.280,172.085,47.781,159.442
C06203=1026.620,360.176,-140.242,172.077,47.780,159.441
C06204=1026.612,359.928,-140.203,172.070,47.779,159.440
C06205=1026.603,359.682,-140.164,172.063,47.779,159.439
C06206=1026.595,359.435,-140.125,172.056,47.779,159.438
C06207=1026.587,359.188,-140.087,172.048,47.778,159.437
C06208=1026.579,358.941,-140.048,172.041,47.777,159.435
C06209=1026.571,358.694,-140.009,172.034,47.777,159.434
C06210=1026.563,358.448,-139.971,172.026,47.776,159.433
C06211=1026.555,358.201,-139.932,172.019,47.776,159.432
C06212=1026.547,357.953,-139.894,172.012,47.775,159.431
C06213=1026.539,357.707,-139.855,172.005,47.774,159.430
C06214=1026.531,357.460,-139.817,171.999,47.774,159.429
C06215=1026.523,357.212,-139.778,171.991,47.773,159.428
C06216=1026.516,356.966,-139.740,171.984,47.773,159.426
C06217=1026.507,356.719,-139.701,171.977,47.773,159.426
C06218=1026.500,356.472,-139.663,171.970,47.772,159.424
C06219=1026.492,356.225,-139.624,171.962,47.771,159.423
C06220=1026.484,355.978,-139.587,171.955,47.771,159.422
C06221=1026.476,355.731,-139.549,171.949,47.770,159.421
C06222=1026.468,355.484,-139.511,171.942,47.770,159.420
C06223=1026.460,355.237,-139.472,171.935,47.769,159.419
C06224=1026.452,354.991,-139.434,171.928,47.769,159.418
C06225=1026.444,354.743,-139.396,171.920,47.769,159.417
C06226=1026.437,354.496,-139.358,171.913,47.769,159.416
C06227=1026.428,354.249,-139.320,171.907,47.768,159.415
C06228=1026.421,354.002,-139.282,171.900,47.768,159.414
C06229=1026.413,353.755,-139.243,171.893,47.768,159.413
C06230=1026.404,353.509,-139.206,171.886,47.767,159.412
C06231=1026.397,353.261,-139.168,171.879,47.767,159.411
C06232=1026.389,353.015,-139.130,171.873,47.766,159.410
C06233=1026.382,352.767,-139.092,171.866,47.766,159.409
C06234=1026.373,352.520,-139.054,171.858,47.766,159.408
C06235=1026.366,352.273,-139.017,171.851,47.766,159.407
C06236=1026.357,352.026,-138.978,171.845,47.765,159.406
C06237=1026.351,351.805,-138.944,171.838,47.765,159.405
C06238=1026.344,351.583,-138.911,171.832,47.765,159.404
C06239=1026.337,351.361,-138.877,171.826,47.764,159.403
C06240=1026.330,351.140,-138.843,171.820,47.764,159.402
C06241=1026.323,350.918,-138.809,171.815,47.764,159.401
C06242=1026.316,350.696,-138.775,171.809,47.764,159.400
C06243=1026.309,350.474,-138.742,171.803,47.763,159.400
C06244=1026.302,350.254,-138.708,171.796,47.763,159.399
C06245=1026.294,350.006,-138.671,171.790,47.763,159.398
C06246=1026.287,349.759,-138.633,171.783,47.763,159.397
C06247=1026.279,349.511,-138.595,171.776,47.763,159.396
C06248=1026.271,349.265,-138.558,171.770,47.762,159.395
C06249=1026.264,349.018,-138.520,171.763,47.762,159.394
C06250=1026.256,348.771,-138.483,171.756,47.762,159.393
C06251=1026.248,348.523,-138.445,171.750,47.762,159.392
C06252=1026.241,348.276,-138.408,171.743,47.762,159.391
C06253=1026.233,348.029,-138.371,171.736,47.762,159.390
C06254=1026.226,347.782,-138.333,171.730,47.762,159.389
C06255=1026.218,347.536,-138.296,171.723,47.762,159.388
C06256=1026.210,347.288,-138.259,171.716,47.762,159.387
C06257=1026.202,347.041,-138.221,171.710,47.761,159.386
C06258=1026.194,346.794,-138.184,171.703,47.762,159.386
C06259=1026.187,346.546,-138.148,171.696,47.762,159.385
C06260=1026.180,346.299,-138.110,171.690,47.761,159.384
C06261=1026.172,346.052,-138.073,171.683,47.761,159.383
C06262=1026.164,345.806,-138.036,171.677,47.762,159.382
C06263=1026.156,345.558,-137.999,171.670,47.761,159.381
C06264=1026.149,345.311,-137.963,171.663,47.761,159.380
C06265=1026.141,345.064,-137.925,171.658,47.762,159.379
C06266=1026.133,344.817,-137.888,171.651,47.761,159.378
C06267=1026.126,344.569,-137.851,171.645,47.761,159.378
C06268=1026.119,344.322,-137.814,171.638,47.762,159.377
C06269=1026.111,344.076,-137.777,171.631,47.761,159.376
C06270=1026.104,343.828,-137.741,171.625,47.762,159.375
C06271=1026.096,343.581,-137.704,171.618,47.762,159.374
C06272=1026.088,343.334,-137.666,171.613,47.762,159.373
C06273=1026.081,343.086,-137.630,171.606,47.762,159.372
C06274=1026.073,342.840,-137.593,171.600,47.762,159.372
C06275=1026.066,342.592,-137.556,171.593,47.762,159.371
C06276=1026.058,342.345,-137.519,171.586,47.762,159.370
C06277=1026.050,342.098,-137.483,171.580,47.762,159.369
C06278=1026.043,341.850,-137.446,171.574,47.763,159.368
C06279=1026.036,341.604,-137.410,171.568,47.763,159.367
C06280=1026.028,341.356,-137.373,171.561,47.763,159.367
C06281=1026.021,341.109,-137.336,171.555,47.763,159.366
C06282=1026.013,340.862,-137.300,171.549,47.763,159.365
C06283=1026.006,340.614,-137.263,171.543,47.763,159.364
C06284=1025.999,340.366,-137.227,171.536,47.763,159.363
C06285=1025.991,340.120,-137.190,171.530,47.764,159.363
C06286=1025.984,339.873,-137.154,171.524,47.764,159.362
C06287=1025.976,339.625,-137.118,171.517,47.764,159.361
C06288=1025.968,339.378,-137.081,171.511,47.764,159.360
C06289=1025.961,339.131,-137.045,171.505,47.765,159.359
C06290=1025.953,338.884,-137.009,171.498,47.765,159.359
C06291=1025.945,338.637,-136.972,171.493,47.765,159.358
C06292=1025.939,338.389,-136.936,171.486,47.766,159.357
C06293=1025.931,338.142,-136.899,171.480,47.766,159.356
C06294=1025.924,337.895,-136.864,171.474,47.767,159.356
C06295=1025.916,337.648,-136.827,171.468,47.767,159.355
C06296=1025.908,337.400,-136.791,171.461,47.767,159.354
C06297=1025.902,337.177,-136.759,171.457,47.767,159.353
C06298=1025.896,336.954,-136.727,171.451,47.767,159.353
C06299=1025.889,336.730,-136.694,171.445,47.768,159.352
C06300=1025.882,336.507,-136.661,171.440,47.768,159.351
C06301=1025.875,336.284,-136.629,171.434,47.769,159.351
C06302=1025.868,336.060,-136.596,171.429,47.769,159.350
C06303=1025.862,335.838,-136.564,171.423,47.769,159.349
C06304=1025.855,335.615,-136.531,171.417,47.769,159.349
C06305=1025.848,335.367,-136.496,171.412,47.770,159.348
C06306=1025.841,335.120,-136.460,171.405,47.771,159.347
C06307=1025.833,334.872,-136.424,171.400,47.771,159.347
C06308=1025.826,334.625,-136.387,171.394,47.771,159.346
C06309=1025.819,334.377,-136.352,171.387,47.772,159.345
C06310=1025.812,334.130,-136.315,171.381,47.772,159.344
C06311=1025.805,333.883,-136.280,171.375,47.772,159.344
C06312=1025.797,333.636,-136.243,171.369,47.773,159.343
C06313=1025.790,333.388,-136.208,171.364,47.773,159.342
C06314=1025.782,333.141,-136.173,171.357,47.774,159.342
C06315=1025.775,332.894,-136.137,171.351,47.774,159.341
C06316=1025.767,332.646,-136.101,171.345,47.775,159.340
C06317=1025.761,332.399,-136.066,171.339,47.775,159.339
C06318=1025.753,332.152,-136.030,171.334,47.776,159.339
C06319=1025.746,331.904,-135.995,171.327,47.777,159.338
C06320=1025.738,331.656,-135.960,171.322,47.777,159.337
C06321=1025.731,331.410,-135.924,171.316,47.778,159.337
C06322=1025.724,331.162,-135.889,171.310,47.778,159.336
C06323=1025.716,330.915,-135.853,171.304,47.779,159.336
C06324=1025.710,330.668,-135.818,171.299,47.779,159.335
C06325=1025.702,330.420,-135.783,171.292,47.780,159.334
C06326=1025.694,330.173,-135.747,171.287,47.781,159.334
C06327=1025.687,329.925,-135.711,171.281,47.781,159.333
C06328=1025.680,329.678,-135.676,171.274,47.782,159.332
C06329=1025.674,329.430,-135.641,171.269,47.783,159.332
C06330=1025.665,329.183,-135.605,171.263,47.783,159.331
C06331=1025.658,328.936,-135.570,171.257,47.784,159.330
C06332=1025.652,328.688,-135.535,171.251,47.784,159.330
C06333=1025.644,328.440,-135.500,171.246,47.785,159.329
C06334=1025.637,328.194,-135.464,171.239,47.786,159.328
C06335=1025.630,327.947,-135.429,171.234,47.787,159.328
C06336=1025.622,327.698,-135.394,171.229,47.787,159.327
C06337=1025.616,327.451,-135.359,171.222,47.788,159.326
C06338=1025.609,327.204,-135.323,171.217,47.789,159.326
C06339=1025.601,326.957,-135.289,171.211,47.790,159.325
C06340=1025.593,326.709,-135.254,171.205,47.791,159.325
C06341=1025.586,326.462,-135.219,171.199,47.791,159.324
C06342=1025.579,326.214,-135.184,171.194,47.792,159.324
C06343=1025.572,325.966,-135.150,171.188,47.793,159.323
C06344=1025.564,325.719,-135.115,171.182,47.794,159.322
C06345=1025.557,325.472,-135.080,171.177,47.795,159.322
C06346=1025.550,325.224,-135.045,171.171,47.795,159.321
C06347=1025.542,324.977,-135.010,171.165,47.797,159.321
C06348=1025.535,324.729,-134.977,171.160,47.797,159.320
C06349=1025.528,324.482,-134.941,171.154,47.798,159.320
C06350=1025.520,324.234,-134.907,171.148,47.799,159.319
C06351=1025.513,323.986,-134.873,171.143,47.800,159.319
C06352=1025.506,323.739,-134.838,171.137,47.801,159.318
C06353=1025.498,323.492,-134.803,171.132,47.802,159.318
C06354=1025.491,323.244,-134.769,171.125,47.803,159.317
C06355=1025.484,322.997,-134.734,171.120,47.804,159.316
C06356=1025.477,322.750,-134.700,171.115,47.805,159.316
C06357=1025.470,322.524,-134.668,171.109,47.805,159.315
C06358=1025.464,322.299,-134.637,171.104,47.806,159.315
C06359=1025.457,322.073,-134.605,171.099,47.807,159.314
C06360=1025.450,321.848,-134.574,171.094,47.808,159.314
C06361=1025.444,321.622,-134.542,171.089,47.809,159.313
C06362=1025.437,321.396,-134.511,171.084,47.810,159.313
C06363=1025.431,321.170,-134.480,171.079,47.811,159.312
C06364=1025.425,320.946,-134.449,171.074,47.811,159.312
C06365=1025.417,320.697,-134.414,171.068,47.812,159.311
C06366=1025.410,320.450,-134.380,171.063,47.814,159.311
C06367=1025.403,320.203,-134.345,171.057,47.815,159.310
C06368=1025.396,319.955,-134.311,171.052,47.816,159.310
C06369=1025.389,319.708,-134.276,171.046,47.817,159.309
C06370=1025.382,319.460,-134.242,171.040,47.818,159.309
C06371=1025.376,319.213,-134.209,171.035,47.819,159.308
C06372=1025.368,318.966,-134.174,171.030,47.820,159.308
C06373=1025.361,318.718,-134.140,171.025,47.821,159.307
C06374=1025.355,318.470,-134.106,171.019,47.821,159.307
C06375=1025.347,318.223,-134.071,171.013,47.823,159.306
C06376=1025.340,317.975,-134.037,171.008,47.824,159.306
C06377=1025.333,317.727,-134.003,171.003,47.825,159.305
C06378=1025.326,317.480,-133.969,170.997,47.826,159.305
C06379=1025.319,317.233,-133.935,170.992,47.827,159.304
C06380=1025.312,316.985,-133.900,170.987,47.828,159.304
C06381=1025.305,316.737,-133.866,170.981,47.830,159.303
C06382=1025.298,316.490,-133.833,170.975,47.831,159.303
C06383=1025.292,316.242,-133.799,170.970,47.831,159.302
C06384=1025.284,315.995,-133.764,170.965,47.833,159.302
C06385=1025.277,315.747,-133.730,170.960,47.834,159.301
C06386=1025.271,315.499,-133.696,170.955,47.835,159.301
C06387=1025.264,315.252,-133.662,170.949,47.836,159.301
C06388=1025.257,315.005,-133.628,170.943,47.838,159.300
C06389=1025.251,314.757,-133.594,170.938,47.839,159.300
C06390=1025.243,314.509,-133.560,170.933,47.840,159.299
C06391=1025.237,314.262,-133.527,170.927,47.841,159.299
C06392=1025.230,314.014,-133.493,170.922,47.842,159.298
C06393=1025.223,313.766,-133.459,170.917,47.843,159.298
C06394=1025.216,313.519,-133.425,170.912,47.845,159.298
C06395=1025.209,313.272,-133.391,170.907,47.845,159.297
C06396=1025.203,313.024,-133.357,170.902,47.847,159.297
C06397=1025.196,312.776,-133.323,170.896,47.848,159.296
C06398=1025.189,312.529,-133.290,170.891,47.849,159.296
C06399=1025.183,312.281,-133.255,170.885,47.850,159.295
C06400=1025.175,312.033,-133.221,170.880,47.852,159.295
C06401=1025.169,311.786,-133.188,170.875,47.853,159.294
C06402=1025.162,311.539,-133.154,170.869,47.854,159.294
C06403=1025.156,311.291,-133.121,170.864,47.855,159.294
C06404=1025.149,311.043,-133.087,170.859,47.857,159.293
C06405=1025.142,310.795,-133.053,170.854,47.858,159.293
C06406=1025.136,310.548,-133.019,170.849,47.859,159.292
C06407=1025.128,310.300,-132.986,170.844,47.861,159.292
C06408=1025.122,310.053,-132.953,170.839,47.862,159.292
C06409=1025.114,309.805,-132.921,170.834,47.864,159.291
C06410=1025.107,309.558,-132.887,170.829,47.865,159.291
C06411=1025.100,309.310,-132.854,170.822,47.866,159.290
C06412=1025.093,309.062,-132.820,170.817,47.868,159.290
C06413=1025.086,308.814,-132.788,170.812,47.869,159.290
C06414=1025.079,308.567,-132.754,170.807,47.871,159.289
C06415=1025.072,308.319,-132.721,170.802,47.872,159.289
C06416=1025.064,308.072,-132.688,170.797,47.873,159.288
C06417=1025.059,307.849,-132.658,170.792,47.875,159.288
C06418=1025.052,307.626,-132.629,170.788,47.876,159.288
C06419=1025.045,307.402,-132.599,170.783,47.878,159.288
C06420=1025.040,307.180,-132.569,170.778,47.879,159.287
C06421=1025.033,306.957,-132.540,170.774,47.881,159.287
C06422=1025.027,306.733,-132.510,170.769,47.882,159.287
C06423=1025.020,306.511,-132.480,170.765,47.883,159.286
C06424=1025.014,306.289,-132.451,170.760,47.885,159.286
C06425=1025.007,306.040,-132.418,170.755,47.886,159.286
C06426=1025.001,305.793,-132.385,170.750,47.888,159.285
C06427=1024.993,305.545,-132.352,170.745,47.889,159.285
C06428=1024.987,305.298,-132.319,170.740,47.891,159.285
C06429=1024.980,305.049,-132.286,170.735,47.892,159.284
C06430=1024.973,304.802,-132.254,170.730,47.894,159.284
C06431=1024.966,304.554,-132.221,170.725,47.896,159.284
C06432=1024.959,304.307,-132.187,170.720,47.897,159.283
C06433=1024.952,304.060,-132.155,170.715,47.899,159.283
C06434=1024.945,303.811,-132.122,170.710,47.900,159.283
C06435=1024.939,303.564,-132.089,170.705,47.902,159.283
C06436=1024.931,303.316,-132.057,170.699,47.904,159.282
C06437=1024.925,303.068,-132.024,170.694,47.905,159.282
C06438=1024.918,302.820,-131.991,170.689,47.907,159.281
C06439=1024.911,302.573,-131.959,170.684,47.908,159.281
C06440=1024.905,302.325,-131.926,170.680,47.910,159.281
C06441=1024.898,302.077,-131.893,170.675,47.912,159.281
C06442=1024.891,301.829,-131.861,170.669,47.913,159.280
C06443=1024.885,301.582,-131.828,170.665,47.916,159.280
C06444=1024.878,301.333,-131.795,170.660,47.917,159.280
C06445=1024.871,301.086,-131.763,170.655,47.918,159.279
C06446=1024.864,300.839,-131.730,170.650,47.921,159.279
C06447=1024.857,300.591,-131.697,170.645,47.922,159.279
C06448=1024.851,300.343,-131.665,170.640,47.923,159.278
C06449=1024.844,300.095,-131.632,170.635,47.926,159.278
C06450=1024.837,299.848,-131.600,170.630,47.927,159.278
C06451=1024.830,299.600,-131.567,170.625,47.928,159.278
C06452=1024.824,299.352,-131.534,170.620,47.931,159.277
C06453=1024.817,299.104,-131.503,170.615,47.932,159.277
C06454=1024.811,298.857,-131.470,170.611,47.934,159.277
C06455=1024.804,298.608,-131.437,170.606,47.936,159.276
C06456=1024.797,298.361,-131.405,170.602,47.937,159.276
C06457=1024.791,298.114,-131.372,170.597,47.939,159.276
C06458=1024.784,297.866,-131.340,170.592,47.941,159.276
C06459=1024.777,297.617,-131.307,170.587,47.942,159.275
C06460=1024.771,297.370,-131.274,170.582,47.944,159.275
C06461=1024.764,297.123,-131.242,170.577,47.946,159.275
C06462=1024.758,296.874,-131.210,170.573,47.948,159.275
C06463=1024.752,296.627,-131.178,170.568,47.950,159.274
C06464=1024.745,296.379,-131.145,170.563,47.952,159.274
C06465=1024.739,296.131,-131.113,170.558,47.953,159.274
C06466=1024.731,295.883,-131.081,170.553,47.955,159.274
C06467=1024.725,295.636,-131.048,170.548,47.957,159.273
C06468=1024.719,295.387,-131.016,170.543,47.959,159.273
C06469=1024.712,295.140,-130.984,170.538,47.960,159.273
C06470=1024.706,294.892,-130.952,170.534,47.962,159.273
C06471=1024.699,294.644,-130.919,170.530,47.964,159.273
C06472=1024.692,294.397,-130.887,170.525,47.966,159.272
C06473=1024.686,294.149,-130.855,170.520,47.968,159.272
C06474=1024.679,293.902,-130.823,170.515,47.969,159.272
C06475=1024.673,293.653,-130.791,170.510,47.971,159.271
C06476=1024.667,293.405,-130.759,170.506,47.973,159.271
C06477=1024.660,293.190,-130.731,170.502,47.975,159.271
C06478=1024.655,292.977,-130.703,170.497,47.977,159.271
C06479=1024.648,292.763,-130.676,170.493,47.978,159.271
C06480=1024.643,292.548,-130.648,170.489,47.980,159.271
C06481=1024.637,292.334,-130.621,170.485,47.981,159.270
C06482=1024.632,292.120,-130.593,170.481,47.984,159.270
C06483=1024.625,291.906,-130.566,170.477,47.985,159.270
C06484=1024.620,291.691,-130.539,170.473,47.987,159.270
C06485=1024.613,291.444,-130.507,170.469,47.989,159.270
C06486=1024.606,291.196,-130.476,170.464,47.991,159.270
C06487=1024.600,290.947,-130.444,170.459,47.993,159.269
C06488=1024.594,290.700,-130.412,170.454,47.995,159.269
C06489=1024.587,290.452,-130.381,170.449,47.997,159.269
C06490=1024.580,290.204,-130.349,170.445,47.999,159.269
C06491=1024.573,289.956,-130.317,170.440,48.001,159.269
C06492=1024.566,289.709,-130.286,170.435,48.003,159.268
C06493=1024.560,289.460,-130.254,170.431,48.005,159.268
C06494=1024.554,289.212,-130.222,170.426,48.008,159.268
C06495=1024.547,288.965,-130.191,170.421,48.010,159.268
C06496=1024.540,288.717,-130.159,170.416,48.012,159.268
C06497=1024.534,288.469,-130.128,170.413,48.014,159.268
C06498=1024.527,288.221,-130.096,170.408,48.016,159.267
C06499=1024.520,287.973,-130.065,170.403,48.018,159.267
C06500=1024.513,287.725,-130.034,170.399,48.020,159.267
C06501=1024.507,287.477,-130.002,170.394,48.023,159.267
C06502=1024.501,287.229,-129.970,170.389,48.025,159.267
C06503=1024.494,286.981,-129.939,170.385,48.027,159.267
C06504=1024.487,286.733,-129.907,170.380,48.029,159.267
C06505=1024.481,286.486,-129.876,170.375,48.031,159.266
C06506=1024.474,286.238,-129.845,170.371,48.033,159.266
C06507=1024.468,285.990,-129.814,170.366,48.035,159.266
C06508=1024.461,285.742,-129.783,170.362,48.038,159.266
C06509=1024.454,285.494,-129.751,170.358,48.040,159.266
C06510=1024.448,285.246,-129.720,170.353,48.042,159.266
C06511=1024.441,284.998,-129.688,170.348,48.044,159.266
C06512=1024.434,284.750,-129.658,170.344,48.047,159.266
C06513=1024.428,284.502,-129.627,170.339,48.049,159.265
C06514=1024.421,284.255,-129.596,170.335,48.051,159.265
C06515=1024.415,284.006,-129.565,170.330,48.053,159.265
C06516=1024.408,283.758,-129.534,170.325,48.056,159.265
C06517=1024.401,283.510,-129.502,170.321,48.058,159.265
C06518=1024.395,283.262,-129.471,170.316,48.060,159.265
C06519=1024.387,283.014,-129.441,170.313,48.063,159.265
C06520=1024.381,282.767,-129.410,170.308,48.065,159.265
C06521=1024.375,282.518,-129.379,170.304,48.067,159.265
C06522=1024.368,282.271,-129.347,170.299,48.070,159.264
C06523=1024.362,282.022,-129.317,170.294,48.072,159.264
C06524=1024.355,281.774,-129.285,170.290,48.074,159.264
C06525=1024.348,281.527,-129.255,170.285,48.077,159.264
C06526=1024.342,281.279,-129.224,170.281,48.079,159.264
C06527=1024.335,281.030,-129.193,170.276,48.081,159.264
C06528=1024.328,280.782,-129.162,170.271,48.084,159.264
C06529=1024.323,280.534,-129.132,170.268,48.086,159.264
C06530=1024.316,280.287,-129.100,170.263,48.088,159.264
C06531=1024.309,280.038,-129.070,170.259,48.091,159.264
C06532=1024.303,279.791,-129.039,170.254,48.093,159.263
C06533=1024.296,279.543,-129.008,170.250,48.096,159.263
C06534=1024.289,279.295,-128.977,170.245,48.098,159.263
C06535=1024.283,279.046,-128.946,170.240,48.101,159.263
C06536=1024.276,278.799,-128.916,170.237,48.102,159.263
C06537=1024.266,278.382,-128.863,170.229,48.107,159.263
C06538=1024.255,277.966,-128.812,170.221,48.111,159.263
C06539=1024.245,277.550,-128.761,170.214,48.115,159.263
C06540=1024.233,277.133,-128.710,170.207,48.119,159.263
C06541=1024.227,276.885,-128.678,170.202,48.121,159.263
C06542=1024.220,276.638,-128.648,170.198,48.124,159.263
C06543=1024.214,276.389,-128.618,170.194,48.127,159.263
C06544=1024.207,276.141,-128.588,170.189,48.129,159.262
C06545=1024.201,275.893,-128.557,170.185,48.131,159.262
C06546=1024.194,275.645,-128.527,170.181,48.134,159.262
C06547=1024.187,275.397,-128.496,170.177,48.137,159.262
C06548=1024.181,275.149,-128.465,170.172,48.139,159.262
C06549=1024.174,274.901,-128.435,170.168,48.142,159.262
C06550=1024.168,274.653,-128.405,170.163,48.145,159.262
C06551=1024.161,274.405,-128.375,170.159,48.147,159.262
C06552=1024.155,274.156,-128.344,170.155,48.149,159.262
C06553=1024.148,273.909,-128.314,170.151,48.152,159.262
C06554=1024.142,273.660,-128.284,170.146,48.155,159.262
C06555=1024.136,273.413,-128.253,170.142,48.158,159.262
C06556=1024.129,273.164,-128.223,170.138,48.160,159.262
C06557=1024.123,272.917,-128.193,170.133,48.162,159.262
C06558=1024.116,272.668,-128.163,170.128,48.165,159.262
C06559=1024.110,272.421,-128.132,170.125,48.168,159.262
C06560=1024.103,272.172,-128.102,170.121,48.170,159.262
C06561=1024.096,271.924,-128.071,170.116,48.173,159.262
C06562=1024.090,271.676,-128.042,170.112,48.176,159.262
C06563=1024.083,271.428,-128.011,170.108,48.179,159.262
C06564=1024.077,271.180,-127.982,170.103,48.181,159.262
C06565=1024.070,270.931,-127.952,170.099,48.184,159.262
C06566=1024.064,270.684,-127.921,170.095,48.187,159.262
C06567=1024.057,270.436,-127.892,170.091,48.189,159.262
C06568=1024.051,270.188,-127.861,170.086,48.192,159.262
C06569=1024.044,269.940,-127.831,170.082,48.194,159.262
C06570=1024.038,269.691,-127.801,170.078,48.197,159.262
C06571=1024.032,269.443,-127.771,170.073,48.201,159.262
C06572=1024.025,269.195,-127.741,170.070,48.203,159.262
C06573=1024.019,268.947,-127.711,170.066,48.206,159.262
C06574=1024.012,268.699,-127.682,170.061,48.209,159.262
C06575=1024.005,268.451,-127.652,170.057,48.211,159.262
C06576=1023.999,268.202,-127.621,170.053,48.214,159.262
C06577=1023.993,267.954,-127.592,170.048,48.217,159.262
C06578=1023.986,267.707,-127.562,170.044,48.220,159.262
C06579=1023.980,267.458,-127.532,170.040,48.222,159.262
C06580=1023.974,267.210,-127.503,170.036,48.225,159.262
C06581=1023.966,266.962,-127.472,170.032,48.228,159.262
C06582=1023.960,266.714,-127.443,170.028,48.231,159.262
C06583=1023.954,266.466,-127.413,170.023,48.234,159.262
C06584=1023.947,266.217,-127.384,170.019,48.237,159.262
C06585=1023.941,265.970,-127.354,170.015,48.239,159.263
C06586=1023.935,265.721,-127.324,170.011,48.242,159.263
C06587=1023.928,265.473,-127.294,170.007,48.245,159.263
C06588=1023.922,265.225,-127.265,170.003,48.248,159.263
C06589=1023.915,264.977,-127.235,169.998,48.251,159.263
C06590=1023.909,264.729,-127.206,169.994,48.254,159.263
C06591=1023.902,264.481,-127.176,169.991,48.257,159.263
C06592=1023.895,264.232,-127.147,169.986,48.260,159.263
C06593=1023.885,263.821,-127.097,169.980,48.265,159.263
C06594=1023.875,263.409,-127.049,169.973,48.269,159.263
C06595=1023.863,262.997,-127.000,169.966,48.274,159.263
C06596=1023.853,262.586,-126.951,169.959,48.279,159.263
C06597=1023.847,262.338,-126.922,169.955,48.282,159.264
C06598=1023.839,262.089,-126.892,169.951,48.285,159.264
C06599=1023.834,261.841,-126.862,169.946,48.288,159.263
C06600=1023.828,261.593,-126.833,169.942,48.291,159.264
C06601=1023.821,261.344,-126.804,169.938,48.294,159.264
C06602=1023.814,261.097,-126.774,169.934,48.296,159.264
C06603=1023.808,260.848,-126.745,169.930,48.300,159.264
C06604=1023.802,260.600,-126.716,169.926,48.303,159.264
C06605=1023.796,260.352,-126.687,169.922,48.306,159.264
C06606=1023.789,260.103,-126.657,169.918,48.309,159.264
C06607=1023.782,259.856,-126.628,169.914,48.312,159.264
C06608=1023.775,259.608,-126.599,169.910,48.315,159.264
C06609=1023.769,259.360,-126.570,169.906,48.318,159.265
C06610=1023.762,259.111,-126.541,169.902,48.322,159.265
C06611=1023.755,258.863,-126.512,169.898,48.325,159.265
C06612=1023.749,258.615,-126.483,169.894,48.328,159.265
C06613=1023.743,258.367,-126.454,169.890,48.331,159.265
C06614=1023.736,258.118,-126.425,169.885,48.334,159.265
C06615=1023.729,257.870,-126.397,169.881,48.338,159.265
C06616=1023.723,257.622,-126.368,169.877,48.341,159.265
C06617=1023.717,257.373,-126.339,169.874,48.344,159.265
C06618=1023.710,257.125,-126.310,169.870,48.347,159.266
C06619=1023.703,256.877,-126.281,169.866,48.350,159.266
C06620=1023.696,256.629,-126.252,169.861,48.353,159.266
C06621=1023.690,256.380,-126.223,169.857,48.357,159.266
C06622=1023.683,256.133,-126.195,169.853,48.360,159.266
C06623=1023.677,255.885,-126.166,169.849,48.363,159.266
C06624=1023.670,255.635,-126.137,169.846,48.366,159.266
C06625=1023.664,255.387,-126.108,169.842,48.369,159.267
C06626=1023.657,255.139,-126.079,169.838,48.373,159.267
C06627=1023.651,254.891,-126.050,169.833,48.376,159.267
C06628=1023.645,254.643,-126.021,169.829,48.379,159.267
C06629=1023.638,254.394,-125.994,169.825,48.383,159.267
C06630=1023.632,254.146,-125.965,169.821,48.386,159.267
C06631=1023.625,253.897,-125.935,169.818,48.389,159.268
C06632=1023.619,253.649,-125.906,169.814,48.392,159.268
C06633=1023.612,253.401,-125.878,169.810,48.395,159.268
C06634=1023.606,253.153,-125.849,169.806,48.399,159.268
C06635=1023.599,252.905,-125.820,169.802,48.402,159.268
C06636=1023.592,252.657,-125.792,169.798,48.406,159.268
C06637=1023.587,252.408,-125.764,169.794,48.408,159.268
C06638=1023.580,252.160,-125.735,169.790,48.412,159.269
C06639=1023.574,251.912,-125.705,169.786,48.415,159.269
C06640=1023.567,251.663,-125.678,169.782,48.419,159.269
C06641=1023.561,251.415,-125.649,169.778,48.422,159.269
C06642=1023.555,251.167,-125.620,169.774,48.425,159.269
C06643=1023.548,250.919,-125.592,169.771,48.429,159.269
C06644=1023.542,250.670,-125.563,169.767,48.432,159.270
C06645=1023.536,250.422,-125.534,169.762,48.435,159.270
C06646=1023.530,250.174,-125.506,169.758,48.438,159.270
C06647=1023.523,249.926,-125.477,169.754,48.442,159.270
C06648=1023.517,249.677,-125.449,169.750,48.445,159.270
C06649=1023.506,249.264,-125.401,169.744,48.451,159.270
C06650=1023.496,248.850,-125.353,169.737,48.457,159.271
C06651=1023.485,248.437,-125.306,169.731,48.462,159.271
C06652=1023.474,248.024,-125.258,169.725,48.468,159.271
C06653=1023.468,247.775,-125.230,169.722,48.471,159.272
C06654=1023.461,247.527,-125.201,169.718,48.474,159.272
C06655=1023.455,247.278,-125.173,169.714,48.478,159.272
C06656=1023.449,247.030,-125.144,169.710,48.481,159.272
C06657=1023.443,246.782,-125.116,169.705,48.485,159.272
C06658=1023.437,246.534,-125.088,169.702,48.488,159.273
C06659=1023.431,246.286,-125.059,169.698,48.491,159.273
C06660=1023.424,246.037,-125.032,169.694,48.495,159.273
C06661=1023.418,245.789,-125.003,169.690,48.498,159.273
C06662=1023.412,245.540,-124.974,169.686,48.502,159.273
C06663=1023.405,245.293,-124.946,169.683,48.505,159.274
C06664=1023.399,245.044,-124.917,169.679,48.508,159.274
C06665=1023.393,244.795,-124.889,169.675,48.512,159.274
C06666=1023.387,244.548,-124.861,169.671,48.515,159.274
C06667=1023.381,244.299,-124.833,169.667,48.519,159.274
C06668=1023.375,244.050,-124.804,169.664,48.523,159.275
C06669=1023.368,243.803,-124.776,169.660,48.526,159.275
C06670=1023.362,243.554,-124.748,169.656,48.530,159.275
C06671=1023.355,243.305,-124.720,169.652,48.533,159.275
C06672=1023.350,243.057,-124.692,169.648,48.537,159.275
C06673=1023.343,242.810,-124.663,169.646,48.540,159.276
C06674=1023.337,242.561,-124.635,169.641,48.544,159.276
C06675=1023.330,242.312,-124.607,169.637,48.547,159.276
C06676=1023.324,242.064,-124.580,169.633,48.551,159.276
C06677=1023.318,241.815,-124.551,169.630,48.555,159.277
C06678=1023.312,241.567,-124.524,169.626,48.558,159.277
C06679=1023.306,241.319,-124.496,169.623,48.562,159.277
C06680=1023.299,241.071,-124.467,169.619,48.565,159.277
C06681=1023.292,240.822,-124.440,169.615,48.569,159.278
C06682=1023.286,240.574,-124.411,169.611,48.573,159.278
C06683=1023.280,240.326,-124.384,169.607,48.576,159.278
C06684=1023.274,240.077,-124.356,169.603,48.580,159.278
C06685=1023.267,239.829,-124.328,169.600,48.583,159.279
C06686=1023.261,239.580,-124.300,169.596,48.587,159.279
C06687=1023.255,239.332,-124.272,169.592,48.591,159.279
C06688=1023.249,239.084,-124.244,169.588,48.594,159.279
C06689=1023.242,238.835,-124.217,169.585,48.599,159.280
C06690=1023.235,238.587,-124.189,169.581,48.602,159.280
C06691=1023.229,238.338,-124.161,169.577,48.606,159.280
C06692=1023.223,238.090,-124.135,169.574,48.609,159.280
C06693=1023.216,237.842,-124.107,169.570,48.613,159.281
C06694=1023.210,237.593,-124.078,169.566,48.617,159.281
C06695=1023.204,237.344,-124.051,169.562,48.621,159.281
C06696=1023.197,237.097,-124.023,169.558,48.625,159.281
C06697=1023.191,236.848,-123.996,169.555,48.629,159.282
C06698=1023.184,236.600,-123.968,169.551,48.632,159.282
C06699=1023.178,236.351,-123.941,169.548,48.636,159.282
C06700=1023.172,236.103,-123.914,169.544,48.640,159.283
C06701=1023.165,235.855,-123.886,169.540,48.644,159.283
C06702=1023.158,235.606,-123.858,169.537,48.648,159.283
C06703=1023.153,235.357,-123.831,169.533,48.651,159.283
C06704=1023.147,235.109,-123.803,169.529,48.655,159.284
C06705=1023.136,234.689,-123.757,169.523,48.662,159.284
C06706=1023.125,234.270,-123.710,169.517,48.668,159.285
C06707=1023.114,233.851,-123.664,169.511,48.674,159.285
C06708=1023.103,233.431,-123.618,169.504,48.682,159.286
C06709=1023.097,233.182,-123.591,169.500,48.685,159.286
C06710=1023.090,232.934,-123.563,169.497,48.689,159.286
C06711=1023.084,232.686,-123.536,169.494,48.693,159.287
C06712=1023.078,232.437,-123.509,169.490,48.697,159.287
C06713=1023.072,232.189,-123.481,169.486,48.701,159.287
C06714=1023.065,231.941,-123.454,169.482,48.705,159.288
C06715=1023.059,231.692,-123.427,169.478,48.708,159.288
C06716=1023.053,231.444,-123.399,169.474,48.713,159.288
C06717=1023.047,231.195,-123.372,169.472,48.716,159.289
C06718=1023.041,230.947,-123.344,169.468,48.721,159.289
C06719=1023.035,230.698,-123.317,169.464,48.724,159.289
C06720=1023.028,230.449,-123.290,169.460,48.728,159.290
C06721=1023.022,230.201,-123.263,169.457,48.732,159.290
C06722=1023.015,229.953,-123.235,169.453,48.737,159.290
C06723=1023.009,229.704,-123.209,169.449,48.741,159.291
C06724=1023.002,229.456,-123.181,169.446,48.744,159.291
C06725=1022.996,229.207,-123.154,169.443,48.748,159.291
C06726=1022.990,228.959,-123.127,169.439,48.752,159.292
C06727=1022.983,228.710,-123.100,169.435,48.756,159.292
C06728=1022.977,228.462,-123.073,169.431,48.760,159.292
C06729=1022.971,228.213,-123.046,169.428,48.765,159.293
C06730=1022.965,227.965,-123.019,169.424,48.769,159.293
C06731=1022.959,227.717,-122.991,169.420,48.773,159.293
C06732=1022.953,227.468,-122.965,169.418,48.777,159.294
C06733=1022.946,227.219,-122.938,169.414,48.780,159.294
C06734=1022.939,226.971,-122.910,169.410,48.784,159.294
C06735=1022.933,226.723,-122.884,169.406,48.789,159.295
C06736=1022.927,226.474,-122.857,169.403,48.793,159.295
C06737=1022.920,226.226,-122.830,169.399,48.797,159.295
C06738=1022.914,225.977,-122.803,169.395,48.801,159.296
C06739=1022.908,225.729,-122.776,169.392,48.806,159.296
C06740=1022.901,225.480,-122.750,169.388,48.810,159.297
C06741=1022.895,225.232,-122.723,169.385,48.814,159.297
C06742=1022.888,224.983,-122.696,169.381,48.818,159.297
C06743=1022.882,224.735,-122.669,169.378,48.822,159.298
C06744=1022.875,224.486,-122.642,169.375,48.826,159.298
C06745=1022.870,224.238,-122.616,169.371,48.831,159.298
C06746=1022.862,223.989,-122.589,169.367,48.835,159.299
C06747=1022.857,223.741,-122.563,169.364,48.839,159.299
C06748=1022.850,223.492,-122.536,169.360,48.843,159.299
C06749=1022.844,223.244,-122.509,169.356,48.848,159.300
C06750=1022.837,222.995,-122.482,169.353,48.852,159.300
C06751=1022.831,222.747,-122.456,169.349,48.856,159.301
C06752=1022.825,222.499,-122.429,169.345,48.860,159.301
C06753=1022.818,222.250,-122.402,169.342,48.865,159.301
C06754=1022.812,222.002,-122.376,169.338,48.869,159.302
C06755=1022.806,221.752,-122.349,169.335,48.873,159.302
C06756=1022.800,221.504,-122.323,169.332,48.877,159.303
C06757=1022.793,221.255,-122.296,169.328,48.882,159.303
C06758=1022.787,221.007,-122.269,169.325,48.886,159.303
C06759=1022.781,220.759,-122.243,169.321,48.890,159.304
C06760=1022.774,220.510,-122.216,169.317,48.894,159.304
C06761=1022.768,220.296,-122.193,169.315,48.898,159.304
C06762=1022.764,220.083,-122.170,169.312,48.902,159.305
C06763=1022.758,219.869,-122.147,169.308,48.905,159.305
C06764=1022.753,219.655,-122.124,169.305,48.909,159.305
C06765=1022.748,219.442,-122.102,169.303,48.913,159.306
C06766=1022.742,219.228,-122.079,169.300,48.916,159.306
C06767=1022.737,219.014,-122.056,169.297,48.920,159.307
C06768=1022.731,218.800,-122.033,169.293,48.924,159.307
C06769=1022.725,218.551,-122.007,169.290,48.929,159.307
C06770=1022.719,218.303,-121.981,169.286,48.933,159.308
C06771=1022.712,218.055,-121.954,169.283,48.938,159.308
C06772=1022.706,217.806,-121.928,169.280,48.941,159.309
C06773=1022.699,217.558,-121.902,169.276,48.946,159.309
C06774=1022.693,217.309,-121.876,169.273,48.950,159.309
C06775=1022.687,217.060,-121.849,169.269,48.955,159.310
C06776=1022.680,216.812,-121.823,169.266,48.959,159.310
C06777=1022.673,216.564,-121.797,169.262,48.964,159.311
C06778=1022.668,216.315,-121.771,169.259,48.968,159.311
C06779=1022.661,216.067,-121.745,169.255,48.973,159.312
C06780=1022.654,215.818,-121.718,169.252,48.978,159.312
C06781=1022.648,215.537,-121.688,169.248,48.983,159.313
C06782=1022.640,215.254,-121.659,169.244,48.988,159.313
C06783=1022.633,214.973,-121.629,169.240,48.993,159.314
C06784=1022.626,214.692,-121.600,169.236,48.998,159.314
C06785=1022.620,214.442,-121.574,169.232,49.002,159.314
C06786=1022.613,214.194,-121.548,169.229,49.007,159.315
C06787=1022.606,213.946,-121.521,169.225,49.011,159.315
C06788=1022.601,213.697,-121.496,169.223,49.016,159.316
C06789=1022.594,213.448,-121.469,169.219,49.020,159.316
C06790=1022.588,213.200,-121.442,169.216,49.025,159.317
C06791=1022.582,212.951,-121.417,169.212,49.030,159.317
C06792=1022.575,212.703,-121.391,169.209,49.034,159.318
C06793=1022.569,212.454,-121.364,169.205,49.039,159.318
C06794=1022.563,212.206,-121.339,169.202,49.043,159.319
C06795=1022.556,211.958,-121.313,169.198,49.048,159.319
C06796=1022.551,211.709,-121.287,169.195,49.052,159.319
C06797=1022.544,211.460,-121.260,169.191,49.057,159.320
C06798=1022.537,211.212,-121.234,169.188,49.062,159.320
C06799=1022.532,210.963,-121.208,169.184,49.066,159.321
C06800=1022.525,210.715,-121.182,169.181,49.071,159.321
C06801=1022.519,210.466,-121.157,169.178,49.075,159.322
C06802=1022.513,210.217,-121.130,169.174,49.080,159.322
C06803=1022.506,209.968,-121.105,169.171,49.084,159.323
C06804=1022.500,209.720,-121.079,169.167,49.089,159.323
C06805=1022.494,209.472,-121.053,169.164,49.094,159.324
C06806=1022.487,209.224,-121.027,169.161,49.098,159.324
C06807=1022.480,208.974,-121.001,169.157,49.103,159.325
C06808=1022.474,208.725,-120.976,169.154,49.107,159.325
C06809=1022.468,208.477,-120.949,169.150,49.112,159.326
C06810=1022.462,208.228,-120.924,169.147,49.117,159.326
C06811=1022.456,207.980,-120.898,169.144,49.122,159.327
C06812=1022.450,207.732,-120.873,169.140,49.126,159.327
C06813=1022.443,207.482,-120.847,169.137,49.131,159.328
C06814=1022.436,207.234,-120.821,169.133,49.136,159.328
C06815=1022.430,206.986,-120.796,169.130,49.141,159.329
C06816=1022.424,206.737,-120.770,169.127,49.146,159.329
C06817=1022.417,206.489,-120.744,169.124,49.151,159.330
C06818=1022.411,206.240,-120.719,169.120,49.155,159.330
C06819=1022.405,205.991,-120.693,169.117,49.160,159.331
C06820=1022.399,205.742,-120.667,169.113,49.165,159.331
C06821=1022.389,205.351,-120.627,169.108,49.172,159.332
C06822=1022.378,204.960,-120.587,169.103,49.180,159.333
C06823=1022.368,204.570,-120.547,169.097,49.188,159.334
C06824=1022.358,204.178,-120.507,169.092,49.195,159.334
C06825=1022.335,203.145,-120.407,168.665,49.098,159.249
C06826=1022.330,202.895,-120.383,168.661,49.104,159.249
C06827=1022.324,202.647,-120.360,168.657,49.110,159.250
C06828=1022.318,202.398,-120.335,168.651,49.116,159.250
C06829=1022.313,202.149,-120.311,168.647,49.121,159.251
C06830=1022.308,201.900,-120.287,168.643,49.127,159.251
C06831=1022.302,201.652,-120.264,168.639,49.133,159.252
C06832=1022.297,201.403,-120.239,168.635,49.138,159.252
C06833=1022.292,201.154,-120.216,168.631,49.144,159.253
C06834=1022.287,200.905,-120.192,168.627,49.150,159.254
C06835=1022.281,200.657,-120.168,168.622,49.156,159.254
C06836=1022.276,200.408,-120.144,168.618,49.162,159.255
C06837=1022.270,200.159,-120.120,168.614,49.167,159.255
C06838=1022.265,199.909,-120.096,168.610,49.173,159.256
C06839=1022.259,199.661,-120.073,168.606,49.179,159.256
C06840=1022.254,199.412,-120.049,168.602,49.185,159.257
C06841=1022.248,199.164,-120.025,168.597,49.191,159.257
C06842=1022.242,198.915,-120.002,168.593,49.197,159.258
C06843=1022.237,198.666,-119.978,168.589,49.203,159.259
C06844=1022.231,198.417,-119.955,168.585,49.209,159.259
C06845=1022.225,198.169,-119.931,168.581,49.215,159.260
C06846=1022.220,197.920,-119.908,168.576,49.221,159.260
C06847=1022.213,197.670,-119.885,168.572,49.227,159.261
C06848=1022.208,197.422,-119.861,168.568,49.233,159.261
C06849=1022.202,197.173,-119.838,168.564,49.239,159.262
C06850=1022.197,196.924,-119.815,168.559,49.244,159.262
C06851=1022.191,196.675,-119.790,168.555,49.250,159.263
C06852=1022.186,196.426,-119.767,168.551,49.256,159.264
C06853=1022.180,196.177,-119.744,168.546,49.262,159.264
C06854=1022.175,195.929,-119.720,168.542,49.268,159.265
C06855=1022.169,195.680,-119.697,168.538,49.274,159.265
C06856=1022.164,195.431,-119.674,168.534,49.279,159.266
C06857=1022.158,195.182,-119.651,168.530,49.285,159.267
C06858=1022.152,194.934,-119.627,168.526,49.291,159.267
C06859=1022.147,194.684,-119.604,168.522,49.297,159.268
C06860=1022.141,194.436,-119.581,168.517,49.303,159.268
C06861=1022.136,194.187,-119.558,168.513,49.309,159.269
C06862=1022.130,193.938,-119.533,168.509,49.315,159.269
C06863=1022.125,193.689,-119.510,168.505,49.321,159.270
C06864=1022.119,193.440,-119.488,168.501,49.327,159.271
C06865=1022.114,193.191,-119.464,168.497,49.333,159.271
C06866=1022.108,192.942,-119.441,168.493,49.339,159.272
C06867=1022.104,192.694,-119.418,168.489,49.345,159.272
C06868=1022.098,192.445,-119.394,168.485,49.351,159.273
C06869=1022.092,192.196,-119.371,168.481,49.356,159.274
C06870=1022.087,191.947,-119.348,168.477,49.362,159.274
C06871=1022.081,191.698,-119.325,168.473,49.368,159.275
C06872=1022.076,191.449,-119.302,168.469,49.374,159.275
C06873=1022.071,191.200,-119.278,168.464,49.380,159.276
C06874=1022.065,190.951,-119.255,168.460,49.386,159.277
C06875=1022.059,190.702,-119.232,168.456,49.392,159.277
C06876=1022.054,190.453,-119.209,168.453,49.399,159.278
C06877=1022.049,190.206,-119.186,168.449,49.405,159.278
C06878=1022.043,189.957,-119.163,168.445,49.411,159.279
C06879=1022.038,189.708,-119.139,168.441,49.417,159.280
C06880=1022.032,189.459,-119.116,168.437,49.423,159.280
C06881=1022.027,189.210,-119.093,168.433,49.428,159.281
C06882=1022.022,188.961,-119.070,168.429,49.434,159.281
C06883=1022.016,188.712,-119.047,168.425,49.440,159.282
C06884=1022.011,188.463,-119.024,168.421,49.446,159.283
C06885=1022.006,188.214,-119.001,168.417,49.452,159.283
C06886=1022.000,187.932,-118.975,168.413,49.459,159.284
C06887=1021.993,187.650,-118.949,168.408,49.465,159.284
C06888=1021.988,187.369,-118.923,168.404,49.472,159.285
C06889=1021.982,187.087,-118.897,168.399,49.479,159.286
C06890=1021.976,186.838,-118.874,168.395,49.485,159.286
C06891=1021.970,186.589,-118.851,168.391,49.491,159.287
C06892=1021.966,186.340,-118.828,168.387,49.497,159.288
C06893=1021.960,186.091,-118.805,168.383,49.503,159.288
C06894=1021.954,185.843,-118.782,168.379,49.508,159.289
C06895=1021.949,185.593,-118.758,168.376,49.514,159.290
C06896=1021.944,185.345,-118.736,168.372,49.520,159.290
C06897=1021.938,185.096,-118.713,168.368,49.526,159.291
C06898=1021.934,184.847,-118.689,168.365,49.533,159.291
C06899=1021.929,184.598,-118.667,168.361,49.538,159.292
C06900=1021.923,184.349,-118.645,168.357,49.544,159.293
C06901=1021.918,184.100,-118.621,168.353,49.550,159.293
C06902=1021.912,183.851,-118.598,168.349,49.556,159.294
C06903=1021.907,183.603,-118.575,168.345,49.562,159.294
C06904=1021.902,183.353,-118.553,168.341,49.568,159.295
C06905=1021.897,183.104,-118.530,168.337,49.574,159.296
C06906=1021.892,182.856,-118.507,168.334,49.580,159.296
C06907=1021.887,182.607,-118.484,168.330,49.586,159.297
C06908=1021.881,182.357,-118.461,168.326,49.592,159.297
C06909=1021.875,182.108,-118.438,168.322,49.598,159.298
C06910=1021.871,181.860,-118.417,168.319,49.604,159.299
C06911=1021.864,181.611,-118.394,168.315,49.610,159.299
C06912=1021.859,181.362,-118.372,168.311,49.616,159.300
C06913=1021.853,181.113,-118.349,168.307,49.623,159.301
C06914=1021.848,180.864,-118.327,168.303,49.629,159.301
C06915=1021.842,180.615,-118.305,168.300,49.635,159.302
C06916=1021.836,180.366,-118.283,168.296,49.641,159.303
C06917=1021.831,180.118,-118.260,168.292,49.647,159.303
C06918=1021.825,179.868,-118.238,168.288,49.654,159.304
C06919=1021.820,179.619,-118.216,168.284,49.660,159.305
C06920=1021.814,179.371,-118.194,168.280,49.666,159.305
C06921=1021.808,179.121,-118.172,168.277,49.672,159.306
C06922=1021.803,178.872,-118.150,168.273,49.678,159.307
C06923=1021.798,178.624,-118.127,168.269,49.685,159.307
C06924=1021.792,178.375,-118.105,168.265,49.691,159.308
C06925=1021.786,178.126,-118.082,168.261,49.697,159.309
C06926=1021.781,177.877,-118.061,168.258,49.704,159.309
C06927=1021.776,177.627,-118.038,168.254,49.710,159.310
C06928=1021.770,177.379,-118.017,168.250,49.716,159.311
C06929=1021.764,177.130,-117.994,168.246,49.722,159.311
C06930=1021.759,176.880,-117.972,168.242,49.728,159.312
C06931=1021.753,176.632,-117.951,168.239,49.735,159.313
C06932=1021.748,176.383,-117.928,168.235,49.741,159.313
C06933=1021.742,176.133,-117.905,168.231,49.747,159.314
C06934=1021.737,175.885,-117.884,168.227,49.753,159.315
C06935=1021.731,175.635,-117.862,168.223,49.759,159.315
C06936=1021.726,175.387,-117.839,168.220,49.766,159.316
C06937=1021.720,175.138,-117.818,168.216,49.772,159.317
C06938=1021.715,174.889,-117.796,168.212,49.778,159.317
C06939=1021.710,174.640,-117.774,168.209,49.784,159.318
C06940=1021.704,174.392,-117.752,168.205,49.790,159.319
C06941=1021.698,174.142,-117.729,168.202,49.797,159.319
C06942=1021.693,173.893,-117.707,168.198,49.803,159.320
C06943=1021.687,173.644,-117.686,168.194,49.809,159.321
C06944=1021.682,173.395,-117.664,168.190,49.816,159.321
C06945=1021.677,173.146,-117.642,168.187,49.822,159.322
C06946=1021.671,172.897,-117.620,168.183,49.828,159.323
C06947=1021.666,172.649,-117.598,168.179,49.834,159.323
C06948=1021.660,172.399,-117.575,168.176,49.840,159.324
C06949=1021.655,172.151,-117.554,168.173,49.847,159.325
C06950=1021.649,171.868,-117.529,168.168,49.854,159.325
C06951=1021.643,171.586,-117.505,168.163,49.861,159.326
C06952=1021.636,171.304,-117.479,168.160,49.867,159.327
C06953=1021.631,171.021,-117.455,168.156,49.875,159.328
C06954=1021.626,170.772,-117.433,168.152,49.881,159.328
C06955=1021.620,170.523,-117.411,168.149,49.887,159.329
C06956=1021.614,170.275,-117.388,168.145,49.893,159.330
C06957=1021.609,170.026,-117.367,168.141,49.899,159.330
C06958=1021.603,169.777,-117.345,168.138,49.906,159.331
C06959=1021.599,169.528,-117.323,168.134,49.912,159.332
C06960=1021.592,169.279,-117.301,168.130,49.918,159.332
C06961=1021.588,169.030,-117.280,168.127,49.924,159.333
C06962=1021.582,168.780,-117.257,168.123,49.930,159.334
C06963=1021.577,168.532,-117.236,168.120,49.936,159.334
C06964=1021.572,168.283,-117.214,168.116,49.943,159.335
C06965=1021.566,168.034,-117.192,168.112,49.949,159.336
C06966=1021.561,167.785,-117.171,168.110,49.955,159.337
C06967=1021.555,167.536,-117.148,168.106,49.961,159.337
C06968=1021.551,167.287,-117.127,168.102,49.967,159.338
C06969=1021.545,167.038,-117.105,168.098,49.974,159.338
C06970=1021.540,166.789,-117.083,168.095,49.980,159.339
C06971=1021.535,166.539,-117.062,168.092,49.987,159.340
C06972=1021.530,166.291,-117.041,168.088,49.993,159.341
C06973=1021.524,166.041,-117.018,168.084,49.999,159.341
C06974=1021.519,165.792,-116.997,168.081,50.005,159.342
C06975=1021.514,165.544,-116.975,168.078,50.011,159.343
C06976=1021.508,165.294,-116.953,168.074,50.017,159.343
C06977=1021.503,165.046,-116.932,168.070,50.024,159.344
C06978=1021.498,164.797,-116.910,168.067,50.029,159.345
C06979=1021.492,164.548,-116.888,168.064,50.036,159.345
C06980=1021.487,164.299,-116.866,168.060,50.042,159.346
C06981=1021.482,164.050,-116.845,168.056,50.048,159.347
C06982=1021.477,163.800,-116.823,168.053,50.055,159.347
C06983=1021.471,163.552,-116.802,168.049,50.061,159.348
C06984=1021.467,163.303,-116.780,168.046,50.067,159.349
C06985=1021.462,163.054,-116.758,168.043,50.073,159.349
C06986=1021.456,162.805,-116.736,168.039,50.079,159.350
C06987=1021.451,162.555,-116.715,168.035,50.085,159.351
C06988=1021.446,162.307,-116.694,168.032,50.092,159.351
C06989=1021.440,162.057,-116.672,168.029,50.097,159.352
C06990=1021.435,161.809,-116.650,168.025,50.104,159.353
C06991=1021.430,161.559,-116.629,168.021,50.110,159.353
C06992=1021.425,161.311,-116.608,168.019,50.116,159.354
C06993=1021.420,161.062,-116.586,168.015,50.123,159.355
C06994=1021.414,160.813,-116.564,168.011,50.129,159.355
C06995=1021.410,160.563,-116.543,168.008,50.134,159.356
C06996=1021.405,160.314,-116.521,168.005,50.141,159.357
C06997=1021.399,160.066,-116.500,168.001,50.147,159.357
C06998=1021.394,159.816,-116.478,167.998,50.153,159.358
C06999=1021.389,159.567,-116.457,167.994,50.160,159.359
C07000=1021.384,159.318,-116.435,167.992,50.165,159.360
C07001=1021.379,159.070,-116.413,167.988,50.171,159.360
C07002=1021.374,158.820,-116.393,167.984,50.178,159.361
C07003=1021.368,158.571,-116.371,167.980,50.184,159.361
C07004=1021.362,158.322,-116.350,167.978,50.191,159.362
C07005=1021.357,158.073,-116.329,167.974,50.197,159.363
C07006=1021.352,157.824,-116.308,167.970,50.203,159.364
C07007=1021.346,157.575,-116.286,167.967,50.210,159.364
C07008=1021.341,157.326,-116.266,167.964,50.216,159.365
C07009=1021.335,157.077,-116.245,167.961,50.222,159.366
C07010=1021.330,156.828,-116.224,167.957,50.229,159.367
C07011=1021.325,156.579,-116.203,167.954,50.235,159.367
C07012=1021.319,156.330,-116.181,167.951,50.242,159.368
C07013=1021.314,156.080,-116.161,167.947,50.248,159.369
C07014=1021.308,155.798,-116.137,167.944,50.255,159.370
C07015=1021.302,155.515,-116.113,167.939,50.262,159.370
C07016=1021.296,155.233,-116.089,167.936,50.270,159.371
C07017=1021.290,154.950,-116.065,167.931,50.277,159.372
C07018=1021.285,154.701,-116.044,167.929,50.283,159.373
C07019=1021.279,154.452,-116.024,167.925,50.289,159.373
C07020=1021.274,154.204,-116.002,167.922,50.296,159.374
C07021=1021.269,153.955,-115.982,167.918,50.302,159.375
C07022=1021.263,153.705,-115.961,167.915,50.308,159.376
C07023=1021.257,153.456,-115.940,167.912,50.315,159.376
C07024=1021.253,153.207,-115.918,167.908,50.321,159.377
C07025=1021.247,152.958,-115.898,167.905,50.328,159.378
C07026=1021.242,152.708,-115.877,167.902,50.334,159.378
C07027=1021.237,152.460,-115.856,167.898,50.341,159.379
C07028=1021.231,152.211,-115.836,167.896,50.347,159.380
C07029=1021.226,151.962,-115.815,167.892,50.353,159.381
C07030=1021.220,151.712,-115.794,167.888,50.360,159.381
C07031=1021.215,151.463,-115.773,167.886,50.366,159.382
C07032=1021.209,151.214,-115.752,167.882,50.372,159.383
C07033=1021.204,150.965,-115.732,167.878,50.379,159.384
C07034=1021.199,150.716,-115.711,167.876,50.385,159.384
C07035=1021.194,150.467,-115.691,167.872,50.392,159.385
C07036=1021.188,150.218,-115.670,167.869,50.398,159.386
C07037=1021.183,149.969,-115.649,167.866,50.404,159.386
C07038=1021.177,149.720,-115.628,167.862,50.411,159.387
C07039=1021.172,149.471,-115.608,167.858,50.417,159.388
C07040=1021.167,149.222,-115.587,167.856,50.423,159.389
C07041=1021.162,148.973,-115.567,167.853,50.430,159.389
C07042=1021.156,148.724,-115.546,167.849,50.436,159.390
C07043=1021.151,148.474,-115.525,167.846,50.443,159.391
C07044=1021.145,148.225,-115.505,167.843,50.449,159.392
C07045=1021.140,147.976,-115.484,167.839,50.456,159.392
C07046=1021.135,147.727,-115.463,167.836,50.462,159.393
C07047=1021.129,147.478,-115.442,167.833,50.468,159.394
C07048=1021.124,147.229,-115.422,167.829,50.475,159.394
C07049=1021.118,146.980,-115.402,167.827,50.481,159.395
C07050=1021.113,146.731,-115.381,167.823,50.487,159.396
C07051=1021.108,146.482,-115.361,167.820,50.494,159.397
C07052=1021.102,146.233,-115.340,167.817,50.501,159.398
C07053=1021.097,145.984,-115.319,167.813,50.507,159.398
C07054=1021.092,145.734,-115.299,167.811,50.513,159.399
C07055=1021.086,145.485,-115.278,167.807,50.520,159.400
C07056=1021.081,145.236,-115.259,167.803,50.526,159.400
C07057=1021.076,144.987,-115.239,167.801,50.533,159.401
C07058=1021.070,144.738,-115.218,167.797,50.539,159.402
C07059=1021.065,144.488,-115.197,167.794,50.546,159.403
C07060=1021.059,144.240,-115.177,167.791,50.552,159.403
C07061=1021.054,143.991,-115.157,167.788,50.559,159.404
C07062=1021.049,143.741,-115.136,167.784,50.565,159.405
C07063=1021.043,143.492,-115.116,167.781,50.571,159.406
C07064=1021.038,143.243,-115.097,167.778,50.578,159.406
C07065=1021.032,142.994,-115.076,167.774,50.585,159.407
C07066=1021.027,142.745,-115.055,167.772,50.591,159.408
C07067=1021.021,142.496,-115.036,167.768,50.597,159.409
C07068=1021.016,142.247,-115.015,167.766,50.604,159.409
C07069=1021.011,141.997,-114.995,167.762,50.611,159.410
C07070=1021.006,141.748,-114.975,167.759,50.617,159.411
C07071=1021.000,141.500,-114.955,167.756,50.623,159.412
C07072=1020.995,141.251,-114.934,167.753,50.630,159.412
C07073=1020.990,141.001,-114.914,167.750,50.636,159.413
C07074=1020.985,140.752,-114.894,167.746,50.643,159.414
C07075=1020.979,140.503,-114.874,167.743,50.649,159.415
C07076=1020.974,140.254,-114.854,167.740,50.655,159.415
C07077=1020.968,140.005,-114.833,167.737,50.662,159.416
C07078=1020.962,139.722,-114.811,167.734,50.670,159.417
C07079=1020.956,139.438,-114.787,167.730,50.676,159.418
C07080=1020.950,139.156,-114.765,167.726,50.684,159.419
C07081=1020.944,138.874,-114.742,167.723,50.691,159.419
C07082=1020.939,138.624,-114.722,167.719,50.698,159.420
C07083=1020.933,138.375,-114.702,167.717,50.704,159.421
C07084=1020.928,138.126,-114.681,167.713,50.710,159.422
C07085=1020.923,137.876,-114.662,167.711,50.717,159.422
C07086=1020.917,137.627,-114.641,167.707,50.724,159.423
C07087=1020.911,137.378,-114.621,167.704,50.731,159.424
C07088=1020.907,137.129,-114.602,167.701,50.736,159.425
C07089=1020.901,136.881,-114.582,167.697,50.743,159.425
C07090=1020.896,136.631,-114.562,167.695,50.750,159.426
C07091=1020.890,136.382,-114.542,167.692,50.756,159.427
C07092=1020.885,136.132,-114.522,167.688,50.763,159.428
C07093=1020.879,135.883,-114.502,167.685,50.769,159.429
C07094=1020.874,135.634,-114.482,167.682,50.776,159.429
C07095=1020.869,135.386,-114.463,167.680,50.782,159.430
C07096=1020.863,135.136,-114.442,167.676,50.789,159.431
C07097=1020.858,134.887,-114.423,167.672,50.795,159.432
C07098=1020.853,134.638,-114.402,167.670,50.802,159.432
C07099=1020.847,134.388,-114.383,167.667,50.809,159.433
C07100=1020.842,134.139,-114.363,167.664,50.815,159.434
C07101=1020.836,133.891,-114.344,167.660,50.821,159.435
C07102=1020.832,133.641,-114.324,167.658,50.828,159.435
C07103=1020.826,133.392,-114.304,167.655,50.835,159.436
C07104=1020.821,133.142,-114.284,167.651,50.842,159.437
C07105=1020.815,132.893,-114.264,167.648,50.847,159.438
C07106=1020.810,132.645,-114.245,167.645,50.854,159.438
C07107=1020.804,132.396,-114.225,167.642,50.861,159.439
C07108=1020.799,132.146,-114.206,167.639,50.867,159.440
C07109=1020.794,131.896,-114.186,167.636,50.873,159.441
C07110=1020.788,131.648,-114.166,167.633,50.880,159.441
C07111=1020.783,131.399,-114.146,167.631,50.887,159.442
C07112=1020.777,131.150,-114.126,167.627,50.893,159.443
C07113=1020.772,130.900,-114.106,167.624,50.899,159.444
C07114=1020.767,130.651,-114.087,167.621,50.906,159.445
C07115=1020.761,130.402,-114.068,167.619,50.913,159.445
C07116=1020.756,130.153,-114.048,167.615,50.919,159.446
C07117=1020.751,129.903,-114.029,167.612,50.925,159.447
C07118=1020.745,129.654,-114.009,167.609,50.932,159.448
C07119=1020.740,129.405,-113.989,167.606,50.939,159.448
C07120=1020.735,129.156,-113.970,167.603,50.946,159.449
C07121=1020.729,128.907,-113.951,167.600,50.953,159.450
C07122=1020.723,128.657,-113.931,167.596,50.959,159.451
C07123=1020.718,128.409,-113.912,167.594,50.965,159.451
C07124=1020.712,128.160,-113.893,167.590,50.972,159.452
C07125=1020.706,127.910,-113.873,167.588,50.979,159.453
C07126=1020.701,127.661,-113.854,167.584,50.985,159.454
C07127=1020.696,127.412,-113.835,167.581,50.992,159.455
C07128=1020.690,127.163,-113.816,167.579,50.999,159.456
C07129=1020.685,126.913,-113.796,167.575,51.006,159.456
C07130=1020.679,126.664,-113.776,167.573,51.012,159.457
C07131=1020.674,126.415,-113.757,167.569,51.018,159.458
C07132=1020.668,126.166,-113.738,167.567,51.025,159.459
C07133=1020.663,125.916,-113.719,167.563,51.032,159.459
C07134=1020.657,125.668,-113.700,167.560,51.039,159.460
C07135=1020.652,125.418,-113.681,167.558,51.045,159.461
C07136=1020.646,125.169,-113.661,167.554,51.052,159.462
C07137=1020.641,124.920,-113.643,167.551,51.058,159.462
C07138=1020.635,124.671,-113.623,167.548,51.065,159.463
C07139=1020.630,124.421,-113.603,167.546,51.071,159.464
C07140=1020.625,124.172,-113.585,167.542,51.078,159.465
C07141=1020.620,123.923,-113.565,167.540,51.085,159.466
C07142=1020.613,123.640,-113.544,167.536,51.093,159.467
C07143=1020.607,123.357,-113.522,167.533,51.100,159.467
C07144=1020.601,123.074,-113.500,167.530,51.107,159.468
C07145=1020.595,122.791,-113.478,167.527,51.115,159.469
